FUNCTION_BLOCK "KistlerPresser _FB"   // FB2300, SCL
{ S7_Optimized_Access := 'FALSE' }
// stored: AutoNumber false, SetENOAutomatically false
   VAR_INPUT
      iHW_ID_Input : HW_SUBMODULE;
      iHW_ID_Output : HW_SUBMODULE;
      iSafetyInterlock : Bool;
      iContinueInterlock : Bool;
      iFltQuit : Bool;
      iSnEnable : Bool;   // True->Send SN
      iJogSpeed : Real;
      iJogMaxForce : Real;
      iCalibForce : Real;
      iXEncReference : Real;
      iReadIdentifier : Any;
      iReadPressData : Any;
      iWriteIdentifier : Any;
      iWritePressData : Any;
      iSpareByte : Array[0..19] of Byte;
   END_VAR
   VAR_OUTPUT
      oFltNo : Word;
      oError : Bool;
      oReady : Bool;
      oRdyAmp : Bool;
      oRdyCmd : Bool;
      oZeroXOk : Bool;
      oSetXRefOk : Bool;
      oHomeOk : Bool;
      oStartCycleOk : Bool;
      oCycleOK : Bool;
      oCycleNOK : Bool;
      oWaitRequest : Bool;
      oInHomePos : Bool;
      oRunSeq : Bool;
      oActProgNo : Int;
      oActLabelID : Int;
      oActSensorPos : Real;
      oActServoPos : Real;
      oActForce : Real;
      oActXEncRefValue : Real;
   END_VAR
   VAR
      ProgNo : Int;
      SelectSeq : Int;
      ZeroX : Bool;
      SetXRef : Bool;
      Homing : Bool;
      StartCycle : Bool;
      ContinueSeq : Bool;
      JogPos : Bool;
      JogNeg : Bool;
      JogPosActive : Bool;
      JogNegActive : Bool;
      SpareByte : Array[0..67] of Byte;
      InputMessages : Struct   // Status Inputs
         StatusBits : Struct
            "MIRROR-START" : Bool;   // Mirrored cycle START
            "MIRROR-TARE-Y" : Bool;   // Mirrored channel Y Tare or Reset Piezo
            "MIRROR-ZERO X" : Bool;   // Mirrored channel X Zeros
            "MIRROR-STEST-X" : Bool;   // Mirrored sensor test for sensor X
            "MIRROR-STEST-Y" : Bool;   // Mirrored sensor test for sensor Y
            "ReservedBit000.5" : Bool;   // Reserved
            "MASTER-MEAS" : Bool;   // Mirrored master measurement
            "INC-ZERO" : Bool;   // Mirrored zeros incremental sensor
            "ReservedBit001.0" : Bool;   // Reserved
            "MIRROR-ACK-ADMIN" : Bool;   // Mirrored acknowledgment with administrative rights (e.g.,corresponding warning, alarm)
            "ReservedBit001.2" : Bool;   // Reserved
            "MIRROR-ACCESS" : Bool;   // MIRROR-ACCESS
            AUTO : Bool;   // Mirrored production mode, no editing of setup is possible
            "STAT-RESET" : Bool;   // Mirrored statistics reset
            "STAT-DISABLE" : Bool;   // Deactivate mirrored statistics
            "TARE-EXTENDED-Y" : Bool;   // Mirrored Ext. channel Y Tare or Reset Piezo (maXYmos NC)
            MP : Byte;   // Mirrored measurement program choice
            "ReservedBit003.0" : Bool;   // Reserved
            "ReservedBit003.1" : Bool;   // Reserved
            "RESET-SN-GENERATOR" : Bool;   // Mirrored resetting of global serial number
            "ReservedBit003.3" : Bool;   // Reserved
            "ReservedBit003.4" : Bool;   // Reserved
            "BREAKETEST-ACTIVE" : Bool;   // Brake test is performed
            "ReservedBit003.6" : Bool;   // Reserved
            "ReservedBit003.7" : Bool;   // Reserved
            UNI : Byte;   // Mirrored input signals of UNI
            ReservedByte005 : Byte;   // Reserved
            READY : Bool;   // Already
            "OK-TOTAL" : Bool;   // Results GOOD
            "NOK-TOTAL" : Bool;   // Results BAD
            "NO-PASS" : Bool;   // NO-PASS exceeded
            "ReservedBit006.4" : Bool;   // Reserved
            "ReservedBit006.5" : Bool;   // Reserved
            WARN : Bool;   // Warning
            ALARM : Bool;   // Alarm
            S1 : Bool;   // Switching signal S1
            S2 : Bool;   // Switching signal S2
            "ReservedBit007.2" : Bool;   // Reserved
            "ReservedBit007.3" : Bool;   // Reserved
            "ReservedBit007.4" : Bool;   // Reserved
            "ReservedBit007.5" : Bool;   // Reserved
            "ReservedBit007.6" : Bool;   // Reserved
            "ReservedBit007.7" : Bool;   // Reserved
            "O-UNI" : Byte;   // Freely configurable output signal
            "DRIVE-ENABLE" : Bool;   // Mirrored enable drive
            "RUN-SEQUENCE" : Bool;   // Mirrored command process of the sequence
            "DRIVE-TO-HOMEPOS" : Bool;   // Mirrored command movement on base setting (MP-specific)
            "DRIVE-TO-REFPOS" : Bool;   // Mirrored command movement to reference position (global)
            "JOG-FW" : Bool;   // Mirrored command jogging forwards
            "JOG-BW" : Bool;   // Mirrored command jogging backwards
            "WAIT-REQUEST" : Bool;   // Output is set through sequence object Wait. Sequence waits for continuation through acknowledgment.
            "BRAKETEST-DONE" : Bool;   // Brake test performed.
            "SEQUENCE-STOPPED" : Bool;   // Sequence/command stopped
            "SEQUENCE-END" : Bool;   // Sequence/command ended
            "ONLINE-EO-NOK" : Bool;   // NOK for online evaluation of a corresponding EOs. Measurement ends.
            "EXT-STOP" : Bool;   // External stop was set in sequence object
            "SEQUENCE-ERROR" : Bool;   // Sequence/command error
            "DRIVE-ENABLED" : Bool;   // Enable drive set (current status of the enable)
            "HOMEPOS-REACHED" : Bool;   // Home position reached (NC joining module is in MP-specific home position)
            "REFPOS-REACHED" : Bool;   // Reference position reached (NC joining module is in global reference position)
            STANDSTILL : Bool;   // Standstill
            "BRAKETEST-REQ" : Bool;   // Brake test required
            "SERVO-WARN" : Bool;   // Warning message on the servo amplifier pending
            "SERVO-ERROR" : Bool;   // Alarm message on the servo amplifier pending
            "SMES-ACTIVE" : Bool;   // Safety status SMES active
            "SMST2-ACTIVE" : Bool;   // Safety status SMST2 active
            "SMM1-ACTIVE" : Bool;   // Safety status SMM1 active
            "USER-MODE-ACTIVE" : Bool;   // Output is active (1) when the monitoring of the control via the monitor (in the menu 'Service/Jog Mode' ... Sequence Mode... Referencing) is directly performed by the operator.
            SEQUENCE : Byte;   // Mirrored selection sequence Main, Sub1 ... 3
            "LABEL-ID" : Byte;   // Index of the cuurent trademark
            "CFG-MP" : Byte;   // Selecting of the measuring program for the transmission of data is intended. This applies to both writing and reading. See note below. If objects are to be interpreted globally, Byte 15.7 must be set.
            "ReservedBit015.0" : Bool;   // Reserved
            "ReservedBit015.1" : Bool;   // Reserved
            "ReservedBit015.2" : Bool;   // Reserved
            "ReservedBit015.3" : Bool;   // Reserved
            "ReservedBit015.4" : Bool;   // Reserved
            "ReservedBit015.5" : Bool;   // Reserved
            "ReservedBit015.6" : Bool;   // Reserved
            "GLOBAL-CFG-MP" : Bool;   // If this bit is set, the telegram data is interpreted as global objects.
            "MIRRIR-CFG-ADR" : Byte;   // Mirror CFG-ADR (up V 1.2.x.)
            "MIRRIR-CFG-LENGTH" : Byte;   // Mirror CFG-LENGTH (up V 1.2.x.)
            "SELECT-PAGE" : Byte;   // Selection of the page that is displayed in the address range from address 20.
            "TRANSMISSION-FAULT" : Bool;   // Error flag for transmission error. This is set upon detection of a transmission error with clearing of the bit ACK.
            ACK : Bool;   // Confirmation flag is set (= 1 byte 19.1) when maXYmos the desired action, which was triggered by the bit strobe executes.After receiving Bit ACK, Bit Strobe can be cleared. With clearing of bit strobe, bit ACK bit is reset.
            "DEVICE-AVAILABLE" : Bool;   // Wenn Bit gesetzt ist, ist das maXYmos Gerät über den Feldbus ansprechbar. Das Bit wird nach dem Gerätestart gesetzt und bleibt im Betrieb dauerhaft erhalten
            "ReservedBit019.3" : Bool;   // Reserved
            "CHANGEDSELECTED-MP" : Bool;   // Change flags of the measurement program changed. Flag isset (= 1) when it is detected that data has been modified in the measurement program since the last measurement. The flag is set after the measurement.
            "ReservedBit019.5" : Bool;   // Reserved
            "CHANGED--GLOBAL" : Bool;   // Change flags of global settings changed. Flag is set (= 1) when it has been recognized that global settings have been changed since the last measurement. Bit is only set if input bit is 19.6 = 0.
            "BACKUP-REQUEST" : Bool;   // Requirement to create a backup on the export server
         END_STRUCT;
         FreelyArea : Struct
            XEncRefValue : Real;
            CurValueX_1 : Real;
            CurValueX_2 : Real;
            CurValueY : Real;
            SerialNnmber { ExternalAccessible := 'False'; ExternalVisible := 'False'; ExternalWritable := 'False'} : Array[36..85] of Byte;
            "pvCurveXMIN-X" : Real;
            "pvCurveXMAX-X" : Real;
            "pvCurveYMIN-Y" : Real;
            "pvCurveYMAX-Y" : Real;
            PressData : Array[86..203] of Byte;
         END_STRUCT;
      END_STRUCT;
      OutputMessages : Struct   // Control Outputs
         ControlBits : Struct
            START : Bool;   // Cycle START
            "TARE-Y" : Bool;   // Channel Y Tare or Reset Piezo
            "ZERO X" : Bool;   // Channel X zeros
            "STEST-X" : Bool;   // Trigger sensor test for sensor X
            "STEST-Y" : Bool;   // Trigger sensor test for sensor Y
            "ReservedBit000.5" : Bool;   // Reserved
            "MASTER-MEAS" : Bool;   // MEAS Master measurement
            "INC-ZERO" : Bool;   // Zeros incremental sensor
            "ReservedBit001.0" : Bool;   // Reserved
            "ACK-ADMIN" : Bool;   // Acknowledgment with Admin rights (e.g., corresponding warning, alarm)
            "ReservedBit001.2" : Bool;   // Reserved
            ACCESS : Bool;   // Allows the PLC to give the operator access rights. The rights group (Setter, Operator, Admin) in effect is set via the protectionPlcLogon object. If ACCESS = 1, the operator can use these rights (does not have to register separately), when ACCESS = 0, this corresponds to a logoff.
            AUTO : Bool;   // Bit AUTO must be set (Byte 1.4 = 1) when the measurement program should be switched on using the PLC fieldbus. With AUTO = 1, the PLC has full control over maXYmo. A manual setup is thus also blocked!
            "STAT-RESET" : Bool;   // Rest statistics
            "STAT-DISABLE" : Bool;   // Deactivate statistics
            "TARE-EXTENDED-Y" : Bool;   // Ext. channel Y Tare or Reset Piezo (maXYmos NC)
            MP : Byte;   // Measurement program selection (see also byte 14 page control input control/config bits).
            "ReservedBit003.0" : Bool;   // Reserved
            "ReservedBit003.1" : Bool;   // Reserved
            "RESET-SN-GENERATOR" : Bool;   // Resetting of counter of global serial number
            "ReservedBit003.3" : Bool;   // Reserved
            "ReservedBit003.4" : Bool;   // Reserved
            "ReservedBit003.5" : Bool;   // Reserved
            "ReservedBit003.6" : Bool;   // Reserved
            "ReservedBit003.7" : Bool;   // Reserved
            UNI : Byte;   // Reserved for freely configurable digital input signals
            ReservedByte005 : Byte;   // Reserved
            ReservedByte006 : Byte;   // Reserved
            ReservedByte007 : Byte;   // Reserved
            ReservedByte008 : Byte;   // Reserved
            "DRIVE-ENABLE" : Bool;   // Release drive
            "RUN-SEQUENCE" : Bool;   // Command sequence has been run
            "DRIVE-TO-HOMEPOS" : Bool;   // Command movement to home position (MP-specific)
            "DRIVE-TO-REFPOS" : Bool;   // Command movement to reference position (global)
            "JOG-FW" : Bool;   // Command jogging forwards
            "JOG-BW" : Bool;   // Command jogging backwards
            "CONTNUEFROM-WAIT" : Bool;   // Continue command sequence after WAIT-REQUEST
            "MANUAL-BRAKETEST" : Bool;   // Perform command manual brake test
            "ReservedBit010.0" : Bool;   // Reserved
            "ReservedBit010.1" : Bool;   // Reserved
            "ReservedBit010.2" : Bool;   // Reserved
            "SEQ-EXT-STOP-REQ" : Bool;   // Externer Stop der Sequenz
            "ReservedBit010.4" : Bool;   // Reserved
            "ReservedBit010.5" : Bool;   // Reserved
            "ReservedBit010.6" : Bool;   // Reserved
            "ReservedBit010.7" : Bool;   // Reserved
            ReservedByte011 : Byte;   // Reserved
            "CURRENT SEQUENCE" : Byte;   // Select sequence main, Sub1 ... 3
            ReservedByte013 : Byte;   // Reserved
            "CFG-MP" : Byte;   // CFP Program number
            "ReservedBit015.0" : Bool;   // Reserved
            "ReservedBit015.1" : Bool;   // Reserved
            "ReservedBit015.2" : Bool;   // Reserved
            "ReservedBit015.3" : Bool;   // Reserved
            "ReservedBit015.4" : Bool;   // Reserved
            "ReservedBit015.5" : Bool;   // Reserved
            "ReservedBit015.6" : Bool;   // Reserved
            "GLOBAL-CFG-MP" : Bool;
            "CFG-ADDRESS" : Byte;
            "CFG-LENGTH" : Byte;
            "SELECT-PAGE" : Byte;
            "SAVE-TO-MP" : Bool;
            STROBE : Bool;
            "ReservedBit019.2" : Bool;   // Reserved
            "ReservedBit019.3" : Bool;   // Reserved
            "RESET-CHANGED-SELECTED-MP" : Bool;
            "ReservedBit019.5" : Bool;   // Reserved
            "RESET-CHANGEDGLOBAL" : Bool;
            "BACKUP-REQUEST" : Bool;
         END_STRUCT;
         FreelyArea : Struct
            XEncRefValue : Real;
            JogSpeed : Real;
            JogMaxForce : Real;
            CalibForce : Real;
            SerialNnmber { ExternalAccessible := 'False'; ExternalVisible := 'False'; ExternalWritable := 'False'} : Array[36..85] of Byte;
            PressData : Array[86..219] of Byte;
         END_STRUCT;
      END_STRUCT;
      Info : Struct
         ProgNo : Byte;
         SelectSeq : Byte;
         SelectPage : Byte;
         CfgAddress : Byte;
         CfgLength : Byte;
         Cancel : Bool;
         ContinueSeq : Bool;
      END_STRUCT;
      SetXRefRise : Bool;
      JogRise : Bool;
      HomingRise : Bool;
      StartCycleRise : Bool;
      FltQuitRise : Bool;
      SetXRefOld : Bool;
      JogOld : Bool;
      HomingOld : Bool;
      StartCycleOld : Bool;
      FltQuitOld : Bool;
      SetXRefAct : Bool;
      JogAct : Bool;
      HomeAct : Bool;
      CycleAct : Bool;
      OrderCount : Int;
      Index : Int;
      "Step" : Array[1..5] of Int;
      Ref_Timer_IN : Bool;
      JogTimer_IN : Bool;
      HomeTimer_IN : Bool;
      SeqTimer_IN : Bool;
      HomeTime : Time;
      SeqTime : Time;
      Ref_Timer { S7_SetPoint := 'True'} : TON_TIME;
      Jog_Timer { S7_SetPoint := 'True'} : TON_TIME;
      Home_Timer { S7_SetPoint := 'True'} : TON_TIME;
      Seq_Timer { S7_SetPoint := 'True'} : TON_TIME;
   END_VAR
   VAR_TEMP
      tmpSource : Byte;
      tmpRetVal : Int;
      pTempPNIOData : Any;
      pTempPressdata : Any;
      pAnyPressdata AT pTempPressdata : Struct
         SyntaxID : Byte;
         DataType : Byte;
         DataCount : Int;
         DBNumber : Word;
         BytePointer : DWord;
      END_STRUCT;
   END_VAR
BEGIN
   (*
   Kistler Presser Control Function Block
   ruhlamat Automation Technologies(Suzhou ) Co.,Ltd
   Copyright(c ) 2016.All rights reserved.
   -------------------------------------------------------------------------------------------
   NAME OF FUNCTION BLOCK:"maXYmosCtrl"
   FAMILY:ruhlamat PSL
   VERSION:V1.1
   AUTHOR:Chaoyao.Zheng
   LAST CHANGE:11.09.2017
   -------------------------------------------------------------------------------------------
   Date Name Activity
   11.09.2017 Chaoyao.Zheng Created(V1.0)
   12.21.2017 Qianfeng.Yang Update(Step7->TIA Portal)
   -------------------------------------------------------------------------------------------
   // F001: MEM not ready
   // F002: IndraDrive not ready
   // F003: User mode is active
   // F004: Order when FB not ready
   // F005: Several orders set at the same time
   // F006: Invalid program number
   // F007: Timeout when homing procedures 
   // F008: Timeout when press-in cycle
   // F009: Timeout data handshake
   // F010: Timeout when set var
   *)
   //Begin
   #pTempPNIOData := #InputMessages;
   #tmpRetVal := DPRD_DAT(LADDR := #iHW_ID_Input,
                          RECORD => #pTempPNIOData);
   IF #tmpRetVal <> 0 THEN
       GOTO Error;
   END_IF;

   #pTempPressdata := #iReadIdentifier;
   IF #pAnyPressdata.DataType = B#16#2 AND #pAnyPressdata.DataCount > 0 THEN
       #tmpRetVal := BLKMOV(SRCBLK := #InputMessages.FreelyArea.SerialNnmber, DSTBLK => #pTempPressdata);
   END_IF;

   #pTempPressdata := #iReadPressData;
   IF #pAnyPressdata.DataType = B#16#2 AND #pAnyPressdata.DataCount > 0 THEN
       #tmpRetVal := BLKMOV(SRCBLK := #InputMessages.FreelyArea.PressData, DSTBLK => #pTempPressdata);
   END_IF;

   #oActXEncRefValue := #InputMessages.FreelyArea.XEncRefValue;
   #oActProgNo := BYTE_TO_INT(#InputMessages.StatusBits.MP);
   #oActLabelID := BYTE_TO_INT(#InputMessages.StatusBits."LABEL-ID");
   #oActSensorPos := #InputMessages.FreelyArea.CurValueX_1;
   #oActServoPos := #InputMessages.FreelyArea.CurValueX_2;
   #oActForce := #InputMessages.FreelyArea.CurValueY;
   #oInHomePos := #InputMessages.StatusBits."HOMEPOS-REACHED";
   #oRunSeq := #InputMessages.StatusBits."RUN-SEQUENCE";
   #JogPosActive := #InputMessages.StatusBits."JOG-FW";
   #JogNegActive := #InputMessages.StatusBits."JOG-BW";

   IF #iSafetyInterlock AND NOT #InputMessages.StatusBits."SMES-ACTIVE" THEN
       #oRdyAmp := #InputMessages.StatusBits."DRIVE-ENABLED";
       #OutputMessages.ControlBits."DRIVE-ENABLE" := TRUE;
   ELSE
       #oRdyAmp := FALSE;
       #OutputMessages.ControlBits."DRIVE-ENABLE" := FALSE;
   END_IF;

   #FltQuitRise := NOT #FltQuitOld AND #iFltQuit;
   #FltQuitOld := #iFltQuit;
   #SetXRefRise := NOT #SetXRefOld AND #SetXRef;
   #SetXRefOld := #SetXRef;
   #HomingRise := NOT #HomingOld AND #Homing;
   #HomingOld := #Homing;
   #JogRise := NOT #JogOld AND (#JogPos OR #JogNeg);
   #JogOld := #JogPos OR #JogNeg;
   #StartCycleRise := NOT #StartCycleOld AND #StartCycle;
   #StartCycleOld := #StartCycle;

   IF #FltQuitRise THEN
       IF #OrderCount = 0 THEN
           #oFltNo := W#16#0000;
       END_IF;
       #OutputMessages.ControlBits."ACK-ADMIN" := TRUE;
   ELSE
       #OutputMessages.ControlBits."ACK-ADMIN" := FALSE;
   END_IF;

   IF NOT #InputMessages.StatusBits."DEVICE-AVAILABLE" OR #InputMessages.StatusBits.ALARM THEN
       IF #oFltNo = W#16#0000 THEN
           #oFltNo := W#16#F001;
       END_IF;
   END_IF;

   IF #InputMessages.StatusBits."SERVO-ERROR" THEN
       IF #oFltNo = W#16#0000 THEN
           #oFltNo := W#16#F002;
       END_IF;
   END_IF;

   IF #InputMessages.StatusBits."USER-MODE-ACTIVE" THEN
       IF #oFltNo = W#16#0000 THEN
           #oFltNo := W#16#F003;
       END_IF;
   END_IF;

   IF #oFltNo = W#16#0000 THEN
       IF #JogRise OR #HomingRise OR #StartCycleRise THEN
           IF NOT #oRdyCmd THEN
               #oFltNo := W#16#F004;
           END_IF;
       END_IF;
   END_IF;

   #OrderCount := 0;
   IF #JogPos OR #JogNeg THEN
       #OrderCount := #OrderCount + 1;
   END_IF;

   IF #Homing THEN
       #OrderCount := #OrderCount + 1;
   END_IF;

   IF #StartCycle THEN
       #OrderCount := #OrderCount + 1;
   END_IF;

   IF #SetXRef THEN
       #OrderCount := #OrderCount + 1;
   END_IF;

   IF #OrderCount > 1 THEN
       IF #oFltNo = W#16#0000 THEN
           #oFltNo := W#16#F005;
       END_IF;
   END_IF;

   IF (#oFltNo = W#16#0000)
   THEN
       IF (#ProgNo < 0) OR
           (#ProgNo > 127)
       THEN
           #oFltNo := W#16#F006;
       END_IF;
   END_IF;

   IF #oFltNo = W#16#0000 THEN
       IF #SelectSeq < 0 OR #SelectSeq > 3 THEN
           #oFltNo := W#16#F006;
       END_IF;
   END_IF;

   // ***********************************************************************
   // Sequence --- SetXRef
   // ***********************************************************************
   #Index := 1;
   IF NOT #SetXRef THEN
       IF #SetXRefAct THEN
           #OutputMessages.ControlBits.STROBE := FALSE;
           #SetXRefAct := FALSE;
       END_IF;
   END_IF;

   IF #oFltNo = W#16#0000 AND #SetXRefRise THEN
       #Info.ProgNo := INT_TO_BYTE(#ProgNo);
       #Info.SelectSeq := INT_TO_BYTE(#SelectSeq);
       #Info.SelectPage := 0;
       #Info.CfgAddress := 0;
       #Info.CfgLength := 4;
       #SetXRefAct := TRUE;
       #oSetXRefOk := FALSE;
       #Step[#Index] := 0;
   END_IF;

   #Ref_Timer_IN := FALSE;
   IF #SetXRefAct THEN
       CASE #Step[#Index] OF
           0:
               #Ref_Timer_IN := FALSE;
               #Step[#Index] := #Step[#Index] + 1;

           1:
               IF #InputMessages.StatusBits.READY THEN
                   #Ref_Timer_IN := FALSE;
                   #OutputMessages.ControlBits."CFG-MP" := #Info.ProgNo;
                   #OutputMessages.ControlBits."SELECT-PAGE" := #Info.SelectPage;
                   #OutputMessages.ControlBits."CFG-ADDRESS" := #Info.CfgAddress;
                   #OutputMessages.ControlBits."CFG-LENGTH" := #Info.CfgLength;
                   #OutputMessages.ControlBits."SAVE-TO-MP" := TRUE;
                   #Step[#Index] := #Step[#Index] + 1;
               ELSE
                   #Ref_Timer_IN := TRUE;
                   IF #Ref_Timer.Q THEN
                       #Ref_Timer_IN := FALSE;
                       #oFltNo := W#16#F011;
                       #Step[#Index] := 99;

                   END_IF;
               END_IF;

           2:
               IF #InputMessages.StatusBits."CFG-MP" = #Info.ProgNo AND #InputMessages.StatusBits."SELECT-PAGE" = #Info.SelectPage AND #InputMessages.StatusBits."MIRRIR-CFG-ADR" = #Info.CfgAddress AND #InputMessages.StatusBits."MIRRIR-CFG-LENGTH" = #Info.CfgLength THEN
                   #Ref_Timer_IN := FALSE;
                   #OutputMessages.ControlBits.STROBE := TRUE;
                   #Step[#Index] := #Step[#Index] + 1;
               ELSE
                   #Ref_Timer_IN := TRUE;
                   IF #Ref_Timer.Q THEN
                       #Ref_Timer_IN := FALSE;
                       #oFltNo := W#16#F012;
                       #Step[#Index] := 99;
                   END_IF;
               END_IF;

           3:
               IF #InputMessages.StatusBits.ACK THEN
                   #Ref_Timer_IN := FALSE;
                   IF #InputMessages.StatusBits."TRANSMISSION-FAULT" THEN
                       #oFltNo := W#16#F013;
                   ELSE
                       #OutputMessages.ControlBits.STROBE := FALSE;
                       #Step[#Index] := 99;
                   END_IF;
               ELSE
                   #Ref_Timer_IN := TRUE;
                   IF #Ref_Timer.Q THEN
                       #Ref_Timer_IN := FALSE;
                       #oFltNo := W#16#F014;
                       #Step[#Index] := 99;
                   END_IF;
               END_IF;

           99:
               #Ref_Timer_IN := FALSE;
               #OutputMessages.ControlBits.STROBE := FALSE;
               #SetXRefAct := FALSE;
               IF #oFltNo = W#16#0000 THEN
                   #oSetXRefOk := TRUE;
               END_IF;

           ELSE
               ;
       END_CASE;
   END_IF;
   #Ref_Timer(IN := #Ref_Timer_IN,
              PT := t#1s);

   // ***********************************************************************
   // Sequence --- Jog Pos/Neg
   // ***********************************************************************
   #Index := 2;
   IF NOT #JogPos AND NOT #JogNeg THEN
       IF #JogAct THEN
           #Info.Cancel := TRUE;
       END_IF;
   END_IF;

   IF #oFltNo = W#16#0000 AND #JogRise THEN
       #Info.ProgNo := INT_TO_BYTE(#ProgNo);
       #Info.SelectSeq := INT_TO_BYTE(#SelectSeq);
       #Info.SelectPage := 0;
       #Info.CfgAddress := 4;
       #Info.CfgLength := 8;
       #JogAct := TRUE;
       #Step[#Index] := 0;
   END_IF;

   #JogTimer_IN := FALSE;
   IF #JogAct THEN
       CASE #Step[#Index] OF
           0:
               #JogTimer_IN := FALSE;
               #Step[#Index] := #Step[#Index] + 1;

           1:
               IF #InputMessages.StatusBits.READY THEN
                   #JogTimer_IN := FALSE;
                   #OutputMessages.ControlBits."CFG-MP" := #Info.ProgNo;
                   #OutputMessages.ControlBits."SELECT-PAGE" := #Info.SelectPage;
                   #OutputMessages.ControlBits."CFG-ADDRESS" := #Info.CfgAddress;
                   #OutputMessages.ControlBits."CFG-LENGTH" := #Info.CfgLength;
                   #OutputMessages.ControlBits."SAVE-TO-MP" := FALSE;
                   #Step[#Index] := #Step[#Index] + 1;
               ELSE
                   #JogTimer_IN := TRUE;
                   IF #Jog_Timer.Q THEN
                       #JogTimer_IN := FALSE;
                       #oFltNo := W#16#F008;
                       #Step[#Index] := 99;
                   END_IF;
               END_IF;

           2:
               IF #InputMessages.StatusBits."CFG-MP" = #Info.ProgNo AND #InputMessages.StatusBits."SELECT-PAGE" = #Info.SelectPage AND #InputMessages.StatusBits."MIRRIR-CFG-ADR" = #Info.CfgAddress AND #InputMessages.StatusBits."MIRRIR-CFG-LENGTH" = #Info.CfgLength THEN
                   #JogTimer_IN := FALSE;
                   #OutputMessages.ControlBits.STROBE := TRUE;
                   #Step[#Index] := #Step[#Index] + 1;
               ELSE
                   #JogTimer_IN := TRUE;
                   IF #Jog_Timer.Q THEN
                       #JogTimer_IN := FALSE;
                       #oFltNo := W#16#F008;
                       #Step[#Index] := 99;
                   END_IF;
               END_IF;

           3:
               IF #InputMessages.StatusBits.ACK THEN
                   #JogTimer_IN := FALSE;
                   IF #InputMessages.StatusBits."TRANSMISSION-FAULT" THEN
                       #oFltNo := W#16#F008;
                   ELSE
                       #OutputMessages.ControlBits.STROBE := FALSE;
                       #Step[#Index] := #Step[#Index] + 1;
                   END_IF;
               ELSE
                   #JogTimer_IN := TRUE;
                   IF #Jog_Timer.Q THEN
                       #JogTimer_IN := FALSE;
                       #oFltNo := W#16#F008;
                       #Step[#Index] := 99;
                   END_IF;
               END_IF;

           4:
               #Step[#Index] := #Step[#Index] + 1;

           5:
               IF #InputMessages.StatusBits."DRIVE-ENABLED" THEN
                   #JogTimer_IN := FALSE;
                   #Step[#Index] := #Step[#Index] + 1;
               ELSE
                   #JogTimer_IN := TRUE;
                   IF #Jog_Timer.Q THEN
                       #JogTimer_IN := FALSE;
                       #oFltNo := W#16#F007;
                       #Step[#Index] := 99;
                   END_IF;
               END_IF;

           6:
               IF #JogPos AND NOT #JogNeg THEN
                   #OutputMessages.ControlBits."JOG-FW" := TRUE;
                   #OutputMessages.ControlBits."JOG-BW" := FALSE;
               ELSIF NOT #JogPos AND #JogNeg THEN
                   #OutputMessages.ControlBits."JOG-FW" := FALSE;
                   #OutputMessages.ControlBits."JOG-BW" := TRUE;
               ELSE
                   #Step[#Index] := 99;
               END_IF;

           99:
               #JogTimer_IN := FALSE;
               #OutputMessages.ControlBits.STROBE := FALSE;
               #OutputMessages.ControlBits."JOG-FW" := FALSE;
               #OutputMessages.ControlBits."JOG-BW" := FALSE;
               #JogAct := FALSE;

           ELSE
               ;

       END_CASE;
   END_IF;
   #Jog_Timer(IN := #JogTimer_IN,
              PT := T#1s);

   // ***********************************************************************
   // Sequence --- Drive to home position
   // ***********************************************************************
   #Index := 3;

   IF NOT #Homing THEN
       #oHomeOk := FALSE;
       IF #HomeAct THEN
           #OutputMessages.ControlBits.STROBE := FALSE;
           #OutputMessages.ControlBits.AUTO := FALSE;
           #OutputMessages.ControlBits."DRIVE-TO-HOMEPOS" := FALSE;
           #OutputMessages.ControlBits."DRIVE-TO-REFPOS" := FALSE;
           #HomeAct := FALSE;
       END_IF;
   END_IF;

   //IF #oFltNo = W#16#0000 AND #HomingRise THEN
   //#InputMessages.StatusBits.READY AND 
   IF #InputMessages.StatusBits.READY AND #HomingRise AND NOT #InputMessages.StatusBits.ALARM AND NOT #InputMessages.StatusBits.WARN THEN
       #Info.ProgNo := INT_TO_BYTE(#ProgNo);
       #HomeAct := TRUE;
       #oHomeOk := FALSE;
       #Step[#Index] := 0;
   END_IF;

   #HomeTimer_IN := FALSE;
   IF #HomeAct THEN
       CASE #Step[#Index] OF
           0:
               #HomeTimer_IN := FALSE;
               #HomeTime := t#1S;
               #Step[#Index] := #Step[#Index] + 1;

           1:
               //  IF #InputMessages.StatusBits.READY THEN
               IF #InputMessages.StatusBits.READY AND NOT #InputMessages.StatusBits.ALARM AND NOT #InputMessages.StatusBits.WARN THEN
                   #HomeTimer_IN := FALSE;
                   #OutputMessages.ControlBits.AUTO := TRUE;
                   #Step[#Index] := #Step[#Index] + 1;
               ELSE
                   #HomeTimer_IN := TRUE;
                   #HomeTime := t#1S;
                   IF #Home_Timer.Q THEN
                       #HomeTimer_IN := FALSE;
                       #oFltNo := W#16#F008;
                       #Step[#Index] := 99;
                   END_IF;
               END_IF;

           2:
               IF #InputMessages.StatusBits.READY AND #InputMessages.StatusBits.AUTO THEN
                   #HomeTimer_IN := FALSE;
                   #OutputMessages.ControlBits.MP := #Info.ProgNo;
                   #Step[#Index] := #Step[#Index] + 1;
               ELSE
                   #HomeTimer_IN := TRUE;
                   #HomeTime := t#1S;
                   IF #Home_Timer.Q THEN
                       #HomeTimer_IN := FALSE;
                       #oFltNo := W#16#F008;
                       #Step[#Index] := 99;
                   END_IF;
               END_IF;

           3:
               IF #InputMessages.StatusBits.MP = #Info.ProgNo THEN
                   #HomeTimer_IN := FALSE;
                   #OutputMessages.ControlBits.AUTO := FALSE;
                   #Step[#Index] := #Step[#Index] + 1;
               ELSE
                   #HomeTimer_IN := TRUE;
                   #HomeTime := t#1S;
                   IF #Home_Timer.Q THEN
                       #HomeTimer_IN := FALSE;
                       #oFltNo := W#16#F008;
                       #Step[#Index] := 99;
                   END_IF;
               END_IF;

           4:
               IF NOT #InputMessages.StatusBits.AUTO THEN
                   #HomeTimer_IN := FALSE;
                   #Step[#Index] := #Step[#Index] + 1;
               ELSE
                   #HomeTimer_IN := TRUE;
                   #HomeTime := t#1S;
                   IF #Home_Timer.Q THEN
                       #HomeTimer_IN := FALSE;
                       #oFltNo := W#16#F008;
                       #Step[#Index] := 99;
                   END_IF;
               END_IF;

           5:
               IF #InputMessages.StatusBits."HOMEPOS-REACHED" THEN
                   #Step[#Index] := 99;
               ELSIF #InputMessages.StatusBits."DRIVE-ENABLED" AND NOT #InputMessages.StatusBits."SEQUENCE-STOPPED" AND NOT #InputMessages.StatusBits."HOMEPOS-REACHED" THEN
                   #HomeTimer_IN := FALSE;
                   #OutputMessages.ControlBits."DRIVE-TO-HOMEPOS" := TRUE;
                   #Step[#Index] := #Step[#Index] + 1;
               ELSE
                   ;
                   #HomeTimer_IN := TRUE;
                   #HomeTime := t#2S;
                   IF #Home_Timer.Q THEN
                       #HomeTimer_IN := FALSE;
                       #oFltNo := W#16#F007;
                       #Step[#Index] := 99;
                   END_IF;
               END_IF;

           6:
               IF #InputMessages.StatusBits."DRIVE-TO-HOMEPOS" THEN
                   #HomeTimer_IN := FALSE;
                   #Step[#Index] := #Step[#Index] + 1;
               ELSE
                   ;
                   #HomeTimer_IN := TRUE;
                   #HomeTime := t#2S;
                   IF #Home_Timer.Q THEN
                       #HomeTimer_IN := FALSE;
                       #oFltNo := W#16#F007;
                       #Step[#Index] := 99;
                   END_IF;
               END_IF;

           7:
               IF #InputMessages.StatusBits."HOMEPOS-REACHED" THEN
                   #HomeTimer_IN := FALSE;
                   #OutputMessages.ControlBits."DRIVE-TO-HOMEPOS" := FALSE;
                   #Step[#Index] := #Step[#Index] + 1;
               ELSE
                   ;
                   #HomeTimer_IN := TRUE;
                   #HomeTime := t#60S;
                   IF #Home_Timer.Q THEN
                       #HomeTimer_IN := FALSE;
                       #oFltNo := W#16#F007;
                       #Step[#Index] := 99;
                   END_IF;
               END_IF;

           8:
               IF NOT #InputMessages.StatusBits."DRIVE-TO-HOMEPOS" THEN
                   #HomeTimer_IN := FALSE;
                   #Step[#Index] := 99;
               ELSE
                   #HomeTimer_IN := TRUE;
                   #HomeTime := t#2S;
                   IF #Home_Timer.Q THEN
                       #HomeTimer_IN := FALSE;
                       #oFltNo := W#16#F007;
                       #Step[#Index] := 99;
                   END_IF;
               END_IF;

           99:
               #HomeTimer_IN := FALSE;
               #OutputMessages.ControlBits.STROBE := FALSE;
               #OutputMessages.ControlBits.AUTO := FALSE;
               #OutputMessages.ControlBits."DRIVE-TO-HOMEPOS" := FALSE;
               #OutputMessages.ControlBits."DRIVE-TO-REFPOS" := FALSE;

               #HomeAct := FALSE;
               IF #oFltNo = W#16#0000 THEN
                   #oHomeOk := TRUE;
               END_IF;

           ELSE
               ;

       END_CASE;
   END_IF;
   #Home_Timer(IN := #HomeTimer_IN,
               PT := #HomeTime);


   // ***********************************************************************
   // Sequence --- Sequence mode
   // ***********************************************************************
   #Index := 4;
   IF NOT #StartCycle THEN
       #oStartCycleOk := FALSE;
       IF #CycleAct THEN
           #OutputMessages.ControlBits.AUTO := FALSE;
           #OutputMessages.ControlBits.STROBE := FALSE;
           #OutputMessages.ControlBits."RUN-SEQUENCE" := FALSE;
           #OutputMessages.ControlBits."CONTNUEFROM-WAIT" := FALSE;
           #CycleAct := FALSE;
       END_IF;
   END_IF;


   IF #oFltNo = W#16#0000 AND #StartCycleRise THEN
       #Info.ProgNo := INT_TO_BYTE(#ProgNo);
       #Info.SelectSeq := INT_TO_BYTE(#SelectSeq);
       #Info.SelectPage := 0;
       #Info.CfgAddress := 16;
       #pTempPressdata := #iWritePressData;
       #Info.CfgLength := INT_TO_BYTE(#pAnyPressdata.DataCount) + 50;
       #CycleAct := TRUE;
       #oStartCycleOk := FALSE;
       #oCycleOK := FALSE;
       #oCycleNOK := FALSE;
       #Step[#Index] := 0;
       #Step[#Index + 1] := 0;
       IF #Info.SelectSeq = 0 THEN
           #tmpRetVal := BLKMOV(SRCBLK := #iWriteIdentifier,
                                DSTBLK => #OutputMessages.FreelyArea.SerialNnmber);
           #tmpRetVal := BLKMOV(SRCBLK := #iWritePressData,
                                DSTBLK => #OutputMessages.FreelyArea.PressData);
       END_IF;
   END_IF;

   #oWaitRequest := #InputMessages.StatusBits."WAIT-REQUEST";
   #OutputMessages.ControlBits."CONTNUEFROM-WAIT" := #ContinueSeq AND #iContinueInterlock;

   #SeqTimer_IN := FALSE;
   IF #CycleAct THEN
       CASE #Step[#Index] OF
           0:
               #SeqTimer_IN := FALSE;
               IF #iSnEnable THEN
                   #Step[#Index] := #Step[#Index] + 1;
               ELSE
                   #Step[#Index] := 5;
               END_IF;

           1:
               IF #InputMessages.StatusBits.READY THEN
                   #SeqTimer_IN := FALSE;
                   #OutputMessages.ControlBits."CFG-MP" := #Info.ProgNo;
                   #OutputMessages.ControlBits."SELECT-PAGE" := #Info.SelectPage;
                   #OutputMessages.ControlBits."CFG-ADDRESS" := #Info.CfgAddress;
                   #OutputMessages.ControlBits."CFG-LENGTH" := #Info.CfgLength;
                   #OutputMessages.ControlBits."SAVE-TO-MP" := FALSE;
                   #Step[#Index] := #Step[#Index] + 1;
               ELSE
                   ;
                   #SeqTimer_IN := TRUE;
                   #SeqTime := T#1S;
                   IF #Seq_Timer.Q THEN
                       #SeqTimer_IN := FALSE;
                       #oFltNo := W#16#F008;
                       #Step[#Index] := 99;
                   END_IF;
               END_IF;

           2:
               IF #InputMessages.StatusBits."CFG-MP" = #Info.ProgNo AND #InputMessages.StatusBits."SELECT-PAGE" = #Info.SelectPage AND #InputMessages.StatusBits."MIRRIR-CFG-ADR" = #Info.CfgAddress AND #InputMessages.StatusBits."MIRRIR-CFG-LENGTH" = #Info.CfgLength THEN
                   #SeqTimer_IN := FALSE;
                   #OutputMessages.ControlBits.STROBE := TRUE;
                   #Step[#Index] := #Step[#Index] + 1;
               ELSE
                   ;
                   #SeqTimer_IN := TRUE;
                   #SeqTime := T#1S;
                   IF #Seq_Timer.Q THEN
                       #SeqTimer_IN := FALSE;
                       #oFltNo := W#16#F008;
                       #Step[#Index] := 99;
                   END_IF;
               END_IF;

           3:
               IF #InputMessages.StatusBits.ACK THEN
                   #SeqTimer_IN := FALSE;
                   IF #InputMessages.StatusBits."TRANSMISSION-FAULT" THEN
                       #oFltNo := W#16#F008;
                   ELSE
                       #OutputMessages.ControlBits.STROBE := FALSE;
                       #Step[#Index] := #Step[#Index] + 1;
                   END_IF;
               ELSE
                   ;
                   #SeqTimer_IN := TRUE;
                   #SeqTime := T#1S;
                   IF #Seq_Timer.Q THEN
                       #SeqTimer_IN := FALSE;
                       #oFltNo := W#16#F008;
                       #Step[#Index] := 99;
                   END_IF;
               END_IF;

           4:
               #Step[#Index] := #Step[#Index] + 1;

           5:
               IF #InputMessages.StatusBits.READY THEN
                   #SeqTimer_IN := FALSE;
                   #OutputMessages.ControlBits.AUTO := TRUE;
                   #Step[#Index] := #Step[#Index] + 1;
               ELSE
                   ;
                   #SeqTimer_IN := TRUE;
                   #SeqTime := T#1S;
                   IF #Seq_Timer.Q THEN
                       #SeqTimer_IN := FALSE;
                       #oFltNo := W#16#F008;
                       #Step[#Index] := 99;
                   END_IF;
               END_IF;

           6:
               IF #InputMessages.StatusBits."DRIVE-ENABLED" AND NOT #InputMessages.StatusBits."SEQUENCE-STOPPED" AND #InputMessages.StatusBits.READY AND #InputMessages.StatusBits.AUTO THEN
                   #SeqTimer_IN := FALSE;
                   #OutputMessages.ControlBits.MP := #Info.ProgNo;
                   #OutputMessages.ControlBits."CURRENT SEQUENCE" := #Info.SelectSeq;
                   #Step[#Index] := #Step[#Index] + 1;
               ELSE
                   ;
                   #SeqTimer_IN := TRUE;
                   #SeqTime := T#1S;
                   IF #Seq_Timer.Q THEN
                       #SeqTimer_IN := FALSE;
                       #oFltNo := W#16#F008;
                       #Step[#Index] := 99;
                   END_IF;
               END_IF;

           7:
               IF #InputMessages.StatusBits.MP = #Info.ProgNo AND #InputMessages.StatusBits.SEQUENCE = #Info.SelectSeq THEN
                   #SeqTimer_IN := FALSE;
                   #OutputMessages.ControlBits."RUN-SEQUENCE" := TRUE;
                   #Step[#Index] := #Step[#Index] + 1;
               ELSE
                   ;
                   #SeqTimer_IN := TRUE;
                   #SeqTime := T#1S;
                   IF #Seq_Timer.Q THEN
                       #SeqTimer_IN := FALSE;
                       #oFltNo := W#16#F008;
                       #Step[#Index] := 99;
                   END_IF;
               END_IF;

           8:
               IF #InputMessages.StatusBits."RUN-SEQUENCE" AND NOT #InputMessages.StatusBits."SEQUENCE-END" AND #InputMessages.StatusBits."DRIVE-ENABLED" AND NOT #InputMessages.StatusBits.WARN AND NOT #InputMessages.StatusBits.ALARM THEN
                   #SeqTimer_IN := FALSE;
                   #Step[#Index] := #Step[#Index] + 1;
               ELSE
                   ;
                   #SeqTimer_IN := TRUE;
                   #SeqTime := T#2S;
                   IF #Seq_Timer.Q THEN
                       #SeqTimer_IN := FALSE;
                       #oFltNo := W#16#F008;
                       #Step[#Index] := 99;
                   END_IF;
               END_IF;

           9:
               IF #InputMessages.StatusBits."SEQUENCE-STOPPED" AND #InputMessages.StatusBits."SEQUENCE-END" THEN
                   #SeqTimer_IN := FALSE;
                   #OutputMessages.ControlBits."RUN-SEQUENCE" := FALSE;
                   #Step[#Index] := #Step[#Index] + 1;
               ELSE
                   ;
                   #SeqTimer_IN := TRUE;
                   #SeqTime := T#20m;
                   IF #Seq_Timer.Q THEN
                       #SeqTimer_IN := FALSE;
                       #oFltNo := W#16#F008;
                       #Step[#Index] := 99;
                   END_IF;
               END_IF;

           10:
               IF NOT #InputMessages.StatusBits."RUN-SEQUENCE" AND NOT #InputMessages.StatusBits."SEQUENCE-STOPPED" THEN
                   #SeqTimer_IN := FALSE;
                   #Step[#Index] := 99;
               ELSE
                   ;
                   #SeqTimer_IN := TRUE;
                   #SeqTime := T#2S;
                   IF #Seq_Timer.Q THEN
                       #SeqTimer_IN := FALSE;
                       #oFltNo := W#16#F008;
                       #Step[#Index] := 99;
                   END_IF;
               END_IF;

           99:
               #SeqTimer_IN := FALSE;
               #OutputMessages.ControlBits.AUTO := FALSE;
               #OutputMessages.ControlBits.STROBE := FALSE;
               #OutputMessages.ControlBits."RUN-SEQUENCE" := FALSE;
               #OutputMessages.ControlBits."CONTNUEFROM-WAIT" := FALSE;
               #CycleAct := FALSE;
               IF #oFltNo = W#16#0000 THEN
                   #oStartCycleOk := TRUE;
               END_IF;
               #tmpSource := B#16#00;
               #tmpRetVal := FILL(BVAL := #tmpSource, BLK => #OutputMessages.FreelyArea.SerialNnmber);
               #tmpRetVal := FILL(BVAL := #tmpSource, BLK => #OutputMessages.FreelyArea.PressData);
           ELSE
               ;
       END_CASE;

       CASE #Step[#Index + 1] OF
           0:
               IF #InputMessages.StatusBits.READY AND #OutputMessages.ControlBits."RUN-SEQUENCE" THEN
                   #Step[#Index + 1] := 1;
               END_IF;

           1:
               IF NOT #InputMessages.StatusBits.READY THEN
                   #Step[#Index + 1] := 2;
               END_IF;

           2:
               IF #InputMessages.StatusBits.READY THEN
               (* Evaluation result *)
                   #oCycleOK := #InputMessages.StatusBits."OK-TOTAL" AND NOT #InputMessages.StatusBits."NOK-TOTAL";
                   #oCycleNOK := NOT #InputMessages.StatusBits."OK-TOTAL" OR #InputMessages.StatusBits."NOK-TOTAL";
                   #Step[#Index + 1] := 99;
               END_IF;

           ELSE
               ;

       END_CASE;
   END_IF;
   #Seq_Timer(IN := #SeqTimer_IN,
              PT := #SeqTime);

   IF #OrderCount <> 1 THEN
       #OutputMessages.ControlBits.AUTO := FALSE;
       #OutputMessages.ControlBits.STROBE := FALSE;
       #OutputMessages.ControlBits."RUN-SEQUENCE" := FALSE;
       #OutputMessages.ControlBits."CONTNUEFROM-WAIT" := FALSE;
       #OutputMessages.ControlBits."DRIVE-TO-HOMEPOS" := FALSE;
       #OutputMessages.ControlBits."DRIVE-TO-REFPOS" := FALSE;
       #OutputMessages.ControlBits."JOG-FW" := FALSE;
       #OutputMessages.ControlBits."JOG-BW" := FALSE;
   END_IF;
   IF #OrderCount = 0 THEN
       #OutputMessages.ControlBits.MP := INT_TO_BYTE(#ProgNo);
   END_IF;
   #oError := #oFltNo <> W#16#0000;
   #oReady := #oFltNo = W#16#000 AND #oRdyAmp;
   #oRdyCmd := #oFltNo = W#16#0000 AND #oRdyAmp AND NOT #JogAct AND NOT #HomeAct AND NOT #CycleAct AND NOT #SetXRefAct AND NOT #JogPos AND NOT #JogNeg AND NOT #Homing AND NOT #StartCycle AND NOT #SetXRef AND NOT #InputMessages.StatusBits."RUN-SEQUENCE";
   IF #oRdyCmd OR #InputMessages.StatusBits."WAIT-REQUEST" THEN
       #OutputMessages.ControlBits."ZERO X" := #ZeroX;
   ELSE
       #OutputMessages.ControlBits."ZERO X" := FALSE;
   END_IF;

   #oZeroXOk := #InputMessages.StatusBits."MIRROR-ZERO X";
   #OutputMessages.FreelyArea.XEncRefValue := #iXEncReference;
   #OutputMessages.FreelyArea.JogSpeed := #iJogSpeed;
   #OutputMessages.FreelyArea.JogMaxForce := #iJogMaxForce;
   #OutputMessages.FreelyArea.CalibForce := #iCalibForce;

   #pTempPNIOData := #OutputMessages;
   #tmpRetVal := DPWR_DAT(LADDR := #iHW_ID_Output,
                          RECORD := #pTempPNIOData);
   IF #tmpRetVal <> 0 THEN
       GOTO Error;
   END_IF;

   //End function block
   ENO := 1;
   RETURN;
   //Error
   Error:
   #oError := 1;
   ENO := 0;
   RETURN;
END_FUNCTION_BLOCK

FUNCTION "Robot" : Void   // FC2400, LAD
{ S7_Optimized_Access := 'TRUE' }
// stored: AutoNumber false, SetENOAutomatically false
   VAR_TEMP   // added for the SCL form of the ladder/FBD networks
      _w1 : Bool;
      _w2 : Bool;
      _w3 : Bool;
      _w4 : Bool;
      _w5 : Bool;
      _w6 : Bool;
   END_VAR
BEGIN

REGION Network 1: 调用机器人1 / Call robot 1
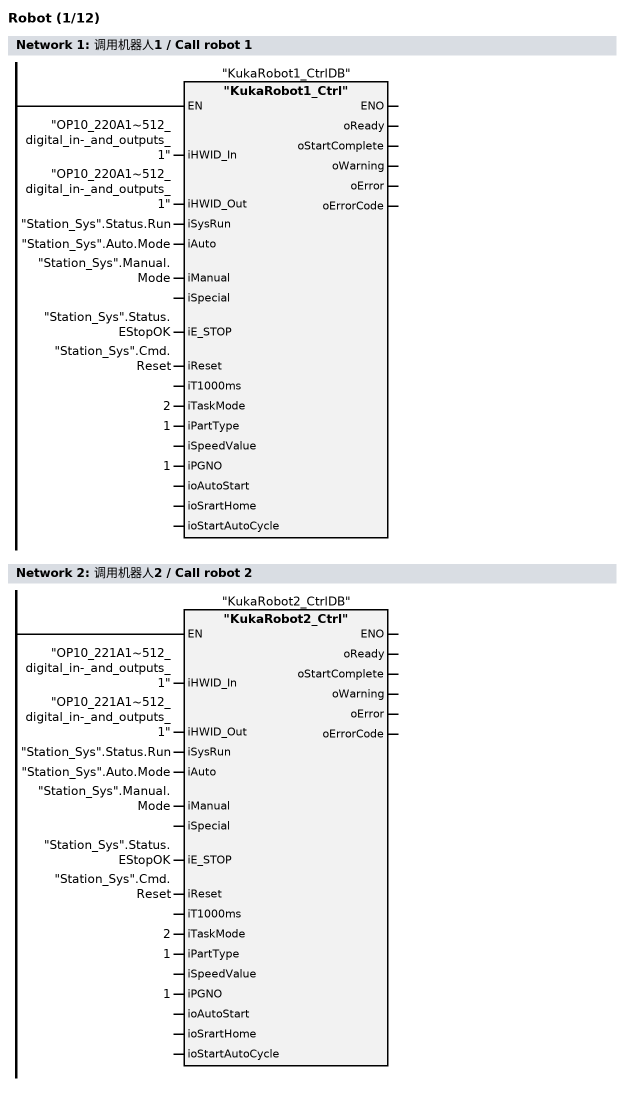
   RUNG wire#powerrail
      "KukaRobot1_CtrlDB"(iHWID_In := "OP10_220A1~512_digital_in-_and_outputs_1", iHWID_Out := "OP10_220A1~512_digital_in-_and_outputs_1", iSysRun := "Station_Sys".Status.Run, iAuto := "Station_Sys".Auto.Mode, iManual := "Station_Sys".Manual.Mode, iSpecial :=, iE_STOP := "Station_Sys".Status.EStopOK, iReset := "Station_Sys".Cmd.Reset, iT1000ms :=, iTaskMode := 2, iPartType := 1, iSpeedValue :=, iPGNO := 1, ioAutoStart :=, ioSrartHome :=, ioStartAutoCycle :=, oReady =>, oStartComplete =>, oWarning =>, oError =>, oErrorCode =>)
   END_RUNG
   // the same network as SCL:
   "KukaRobot1_CtrlDB"(iHWID_In := "OP10_220A1~512_digital_in-_and_outputs_1",   // "KukaRobot1_Ctrl"
                       iHWID_Out := "OP10_220A1~512_digital_in-_and_outputs_1",
                       iSysRun := "Station_Sys".Status.Run,
                       iAuto := "Station_Sys".Auto.Mode,
                       iManual := "Station_Sys".Manual.Mode,
                       iE_STOP := "Station_Sys".Status.EStopOK,
                       iReset := "Station_Sys".Cmd.Reset,
                       iTaskMode := 2,
                       iPartType := 1,
                       iPGNO := 1);
END_REGION

REGION Network 2: 调用机器人2 / Call robot 2
   RUNG wire#powerrail
      "KukaRobot2_CtrlDB"(iHWID_In := "OP10_221A1~512_digital_in-_and_outputs_1", iHWID_Out := "OP10_221A1~512_digital_in-_and_outputs_1", iSysRun := "Station_Sys".Status.Run, iAuto := "Station_Sys".Auto.Mode, iManual := "Station_Sys".Manual.Mode, iSpecial :=, iE_STOP := "Station_Sys".Status.EStopOK, iReset := "Station_Sys".Cmd.Reset, iT1000ms :=, iTaskMode := 2, iPartType := 1, iSpeedValue :=, iPGNO := 1, ioAutoStart :=, ioSrartHome :=, ioStartAutoCycle :=, oReady =>, oStartComplete =>, oWarning =>, oError =>, oErrorCode =>)
   END_RUNG
   // the same network as SCL:
   "KukaRobot2_CtrlDB"(iHWID_In := "OP10_221A1~512_digital_in-_and_outputs_1",   // "KukaRobot2_Ctrl"
                       iHWID_Out := "OP10_221A1~512_digital_in-_and_outputs_1",
                       iSysRun := "Station_Sys".Status.Run,
                       iAuto := "Station_Sys".Auto.Mode,
                       iManual := "Station_Sys".Manual.Mode,
                       iE_STOP := "Station_Sys".Status.EStopOK,
                       iReset := "Station_Sys".Cmd.Reset,
                       iTaskMode := 2,
                       iPartType := 1,
                       iPGNO := 1);
END_REGION

REGION Network 3: 调用机器人3 / Call robot 3
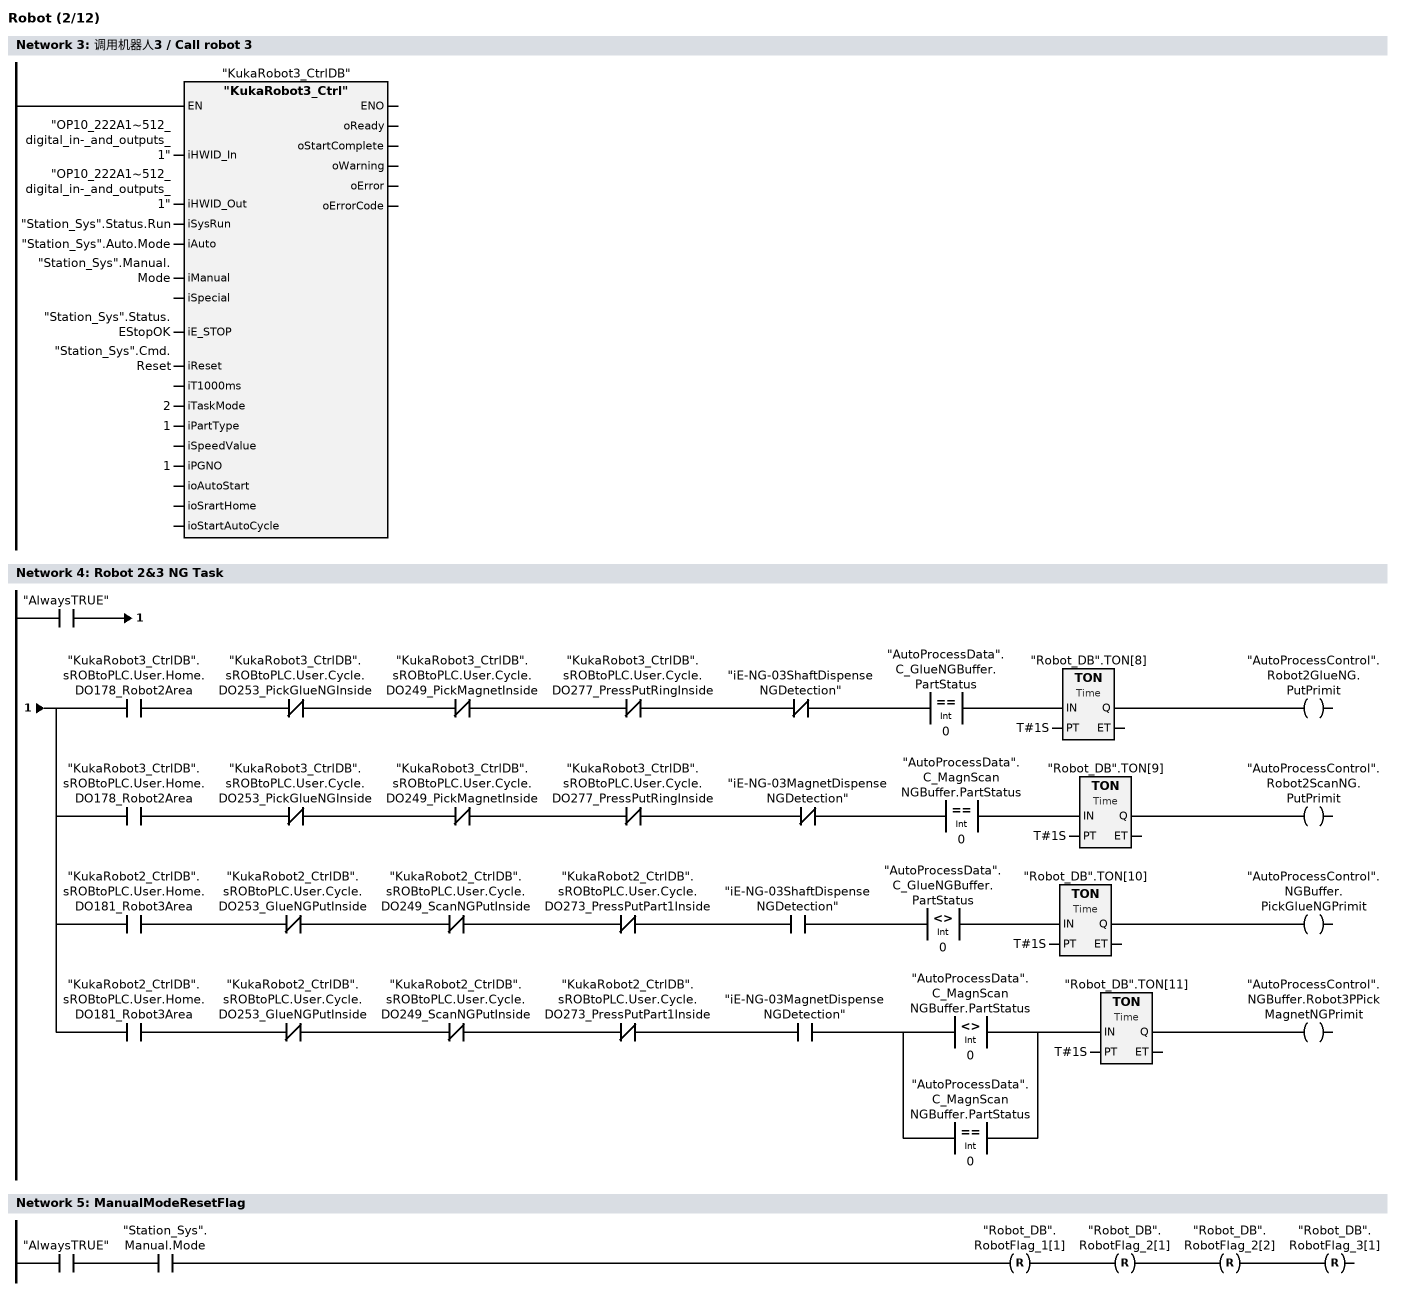
   RUNG wire#powerrail
      "KukaRobot3_CtrlDB"(iHWID_In := "OP10_222A1~512_digital_in-_and_outputs_1", iHWID_Out := "OP10_222A1~512_digital_in-_and_outputs_1", iSysRun := "Station_Sys".Status.Run, iAuto := "Station_Sys".Auto.Mode, iManual := "Station_Sys".Manual.Mode, iSpecial :=, iE_STOP := "Station_Sys".Status.EStopOK, iReset := "Station_Sys".Cmd.Reset, iT1000ms :=, iTaskMode := 2, iPartType := 1, iSpeedValue :=, iPGNO := 1, ioAutoStart :=, ioSrartHome :=, ioStartAutoCycle :=, oReady =>, oStartComplete =>, oWarning =>, oError =>, oErrorCode =>)
   END_RUNG
   // the same network as SCL:
   "KukaRobot3_CtrlDB"(iHWID_In := "OP10_222A1~512_digital_in-_and_outputs_1",   // "KukaRobot3_Ctrl"
                       iHWID_Out := "OP10_222A1~512_digital_in-_and_outputs_1",
                       iSysRun := "Station_Sys".Status.Run,
                       iAuto := "Station_Sys".Auto.Mode,
                       iManual := "Station_Sys".Manual.Mode,
                       iE_STOP := "Station_Sys".Status.EStopOK,
                       iReset := "Station_Sys".Cmd.Reset,
                       iTaskMode := 2,
                       iPartType := 1,
                       iPGNO := 1);
END_REGION

REGION Network 4: Robot 2&3 NG Task
   RUNG wire#powerrail
      Contact( "AlwaysTRUE" )
      wire#w1
      Contact( "KukaRobot3_CtrlDB".sROBtoPLC.User.Home.DO178_Robot2Area )
      I_Contact( "KukaRobot3_CtrlDB".sROBtoPLC.User.Cycle.DO253_PickGlueNGInside )
      I_Contact( "KukaRobot3_CtrlDB".sROBtoPLC.User.Cycle.DO249_PickMagnetInside )
      I_Contact( "KukaRobot3_CtrlDB".sROBtoPLC.User.Cycle.DO277_PressPutRingInside )
      I_Contact( "iE-NG-03ShaftDispenseNGDetection" )
      { S7_Templates := "SrcType := Int" } EQ_Contact(in1 := "AutoProcessData".C_GlueNGBuffer.PartStatus, in2 := 0)
      { S7_Templates := "time_type := Time" } "Robot_DB".TON[8].TON(pt := T#1S, et =>)
      Coil( "AutoProcessControl".Robot2GlueNG.PutPrimit )
   END_RUNG
   RUNG wire#w1
      Contact( "KukaRobot3_CtrlDB".sROBtoPLC.User.Home.DO178_Robot2Area )
      I_Contact( "KukaRobot3_CtrlDB".sROBtoPLC.User.Cycle.DO253_PickGlueNGInside )
      I_Contact( "KukaRobot3_CtrlDB".sROBtoPLC.User.Cycle.DO249_PickMagnetInside )
      I_Contact( "KukaRobot3_CtrlDB".sROBtoPLC.User.Cycle.DO277_PressPutRingInside )
      I_Contact( "iE-NG-03MagnetDispenseNGDetection" )
      { S7_Templates := "SrcType := Int" } EQ_Contact(in1 := "AutoProcessData".C_MagnScanNGBuffer.PartStatus, in2 := 0)
      { S7_Templates := "time_type := Time" } "Robot_DB".TON[9].TON(pt := T#1S, et =>)
      Coil( "AutoProcessControl".Robot2ScanNG.PutPrimit )
   END_RUNG
   RUNG wire#w1
      Contact( "KukaRobot2_CtrlDB".sROBtoPLC.User.Home.DO181_Robot3Area )
      I_Contact( "KukaRobot2_CtrlDB".sROBtoPLC.User.Cycle.DO253_GlueNGPutInside )
      I_Contact( "KukaRobot2_CtrlDB".sROBtoPLC.User.Cycle.DO249_ScanNGPutInside )
      I_Contact( "KukaRobot2_CtrlDB".sROBtoPLC.User.Cycle.DO273_PressPutPart1Inside )
      Contact( "iE-NG-03ShaftDispenseNGDetection" )
      { S7_Templates := "SrcType := Int" } NE_Contact(in1 := "AutoProcessData".C_GlueNGBuffer.PartStatus, in2 := 0)
      { S7_Templates := "time_type := Time" } "Robot_DB".TON[10].TON(pt := T#1S, et =>)
      Coil( "AutoProcessControl".NGBuffer.PickGlueNGPrimit )
   END_RUNG
   RUNG wire#w1
      Contact( "KukaRobot2_CtrlDB".sROBtoPLC.User.Home.DO181_Robot3Area )
      I_Contact( "KukaRobot2_CtrlDB".sROBtoPLC.User.Cycle.DO253_GlueNGPutInside )
      I_Contact( "KukaRobot2_CtrlDB".sROBtoPLC.User.Cycle.DO249_ScanNGPutInside )
      I_Contact( "KukaRobot2_CtrlDB".sROBtoPLC.User.Cycle.DO273_PressPutPart1Inside )
      Contact( "iE-NG-03MagnetDispenseNGDetection" )
      wire#w2
      { S7_Templates := "SrcType := Int" } NE_Contact(in1 := "AutoProcessData".C_MagnScanNGBuffer.PartStatus, in2 := 0)
      wire#w3
      { S7_Templates := "time_type := Time" } "Robot_DB".TON[11].TON(pt := T#1S, et =>)
      Coil( "AutoProcessControl".NGBuffer.Robot3PPickMagnetNGPrimit )
   END_RUNG
   RUNG wire#w2
      { S7_Templates := "SrcType := Int" } EQ_Contact(in1 := "AutoProcessData".C_MagnScanNGBuffer.PartStatus, in2 := 0)
   END_RUNG wire#w3
   // the same network as SCL:
   "Robot_DB".TON[8].TON(IN := "AlwaysTRUE" AND "KukaRobot3_CtrlDB".sROBtoPLC.User.Home.DO178_Robot2Area AND NOT "KukaRobot3_CtrlDB".sROBtoPLC.User.Cycle.DO253_PickGlueNGInside AND NOT "KukaRobot3_CtrlDB".sROBtoPLC.User.Cycle.DO249_PickMagnetInside AND NOT "KukaRobot3_CtrlDB".sROBtoPLC.User.Cycle.DO277_PressPutRingInside AND NOT "iE-NG-03ShaftDispenseNGDetection" AND ("AutoProcessData".C_GlueNGBuffer.PartStatus = 0),
                         PT := T#1S);
   "AutoProcessControl".Robot2GlueNG.PutPrimit := "Robot_DB".TON[8].Q;
   "Robot_DB".TON[9].TON(IN := "AlwaysTRUE" AND "KukaRobot3_CtrlDB".sROBtoPLC.User.Home.DO178_Robot2Area AND NOT "KukaRobot3_CtrlDB".sROBtoPLC.User.Cycle.DO253_PickGlueNGInside AND NOT "KukaRobot3_CtrlDB".sROBtoPLC.User.Cycle.DO249_PickMagnetInside AND NOT "KukaRobot3_CtrlDB".sROBtoPLC.User.Cycle.DO277_PressPutRingInside AND NOT "iE-NG-03MagnetDispenseNGDetection" AND ("AutoProcessData".C_MagnScanNGBuffer.PartStatus = 0),
                         PT := T#1S);
   "AutoProcessControl".Robot2ScanNG.PutPrimit := "Robot_DB".TON[9].Q;
   "Robot_DB".TON[10].TON(IN := "AlwaysTRUE" AND "KukaRobot2_CtrlDB".sROBtoPLC.User.Home.DO181_Robot3Area AND NOT "KukaRobot2_CtrlDB".sROBtoPLC.User.Cycle.DO253_GlueNGPutInside AND NOT "KukaRobot2_CtrlDB".sROBtoPLC.User.Cycle.DO249_ScanNGPutInside AND NOT "KukaRobot2_CtrlDB".sROBtoPLC.User.Cycle.DO273_PressPutPart1Inside AND "iE-NG-03ShaftDispenseNGDetection" AND ("AutoProcessData".C_GlueNGBuffer.PartStatus <> 0),
                          PT := T#1S);
   "AutoProcessControl".NGBuffer.PickGlueNGPrimit := "Robot_DB".TON[10].Q;
   "Robot_DB".TON[11].TON(IN := "AlwaysTRUE" AND "KukaRobot2_CtrlDB".sROBtoPLC.User.Home.DO181_Robot3Area AND NOT "KukaRobot2_CtrlDB".sROBtoPLC.User.Cycle.DO253_GlueNGPutInside AND NOT "KukaRobot2_CtrlDB".sROBtoPLC.User.Cycle.DO249_ScanNGPutInside AND NOT "KukaRobot2_CtrlDB".sROBtoPLC.User.Cycle.DO273_PressPutPart1Inside AND "iE-NG-03MagnetDispenseNGDetection" AND (("AutoProcessData".C_MagnScanNGBuffer.PartStatus <> 0) OR ("AutoProcessData".C_MagnScanNGBuffer.PartStatus = 0)),
                          PT := T#1S);
   "AutoProcessControl".NGBuffer.Robot3PPickMagnetNGPrimit := "Robot_DB".TON[11].Q;
END_REGION

REGION Network 5: ManualModeResetFlag
   RUNG wire#powerrail
      Contact( "AlwaysTRUE" )
      Contact( "Station_Sys".Manual.Mode )
      R_Coil( "Robot_DB".RobotFlag_1[1] )
      R_Coil( "Robot_DB".RobotFlag_2[1] )
      R_Coil( "Robot_DB".RobotFlag_2[2] )
      R_Coil( "Robot_DB".RobotFlag_3[1] )
   END_RUNG
   // the same network as SCL:
   IF "AlwaysTRUE" AND "Station_Sys".Manual.Mode THEN
       "Robot_DB".RobotFlag_1[1] := FALSE;
       "Robot_DB".RobotFlag_2[1] := FALSE;
       "Robot_DB".RobotFlag_2[2] := FALSE;
       "Robot_DB".RobotFlag_3[1] := FALSE;
   END_IF;
END_REGION

REGION Network 6 (SCL): LoadNG传感器 / Loadng sensor
   //NG1
   "KukaRobot1_CtrlDB".sPLCtoROB.User.Home.DI177_NG1_1:="Robot_DB".LoadNG_1[1] := NOT  "iE1-UnloadingShaftPressNG_5";
   "KukaRobot1_CtrlDB".sPLCtoROB.User.Home.DI178_NG1_2:="Robot_DB".LoadNG_1[2] := NOT  "iE1-UnloadingShaftPressNG_4";
   "KukaRobot1_CtrlDB".sPLCtoROB.User.Home.DI179_NG1_3:="Robot_DB".LoadNG_1[3] := NOT  "iE1-UnloadingShaftPressNG_3";
   "KukaRobot1_CtrlDB".sPLCtoROB.User.Home.DI180_NG1_4:="Robot_DB".LoadNG_1[4] := NOT  "iE1-UnloadingShaftPressNG_2";
   "KukaRobot1_CtrlDB".sPLCtoROB.User.Home.DI181_NG1_5:="Robot_DB".LoadNG_1[5] := NOT  "iE1-UnloadingShaftPressNG_1";

   //NG2
   "KukaRobot1_CtrlDB".sPLCtoROB.User.Home.DI182_NG2_1:="Robot_DB".LoadNG_2[1] := NOT  "iE1-UnloadingShaftScanNG_5";
   "KukaRobot1_CtrlDB".sPLCtoROB.User.Home.DI183_NG2_2:="Robot_DB".LoadNG_2[2] := NOT  "iE1-UnloadingShaftScanNG_4";
   "KukaRobot1_CtrlDB".sPLCtoROB.User.Home.DI184_NG2_3:="Robot_DB".LoadNG_2[3] := NOT  "iE1-UnloadingShaftScanNG_3";
   "KukaRobot1_CtrlDB".sPLCtoROB.User.Home.DI185_NG2_4:="Robot_DB".LoadNG_2[4] := NOT  "iE1-UnloadingShaftScanNG_2";
   "KukaRobot1_CtrlDB".sPLCtoROB.User.Home.DI186_NG2_5:="Robot_DB".LoadNG_2[5] := NOT  "iE1-UnloadingShaftScanNG_1";

   //NG3
   "KukaRobot1_CtrlDB".sPLCtoROB.User.Home.DI187_NG3_1:="Robot_DB".LoadNG_3[1] := NOT  "iE1-UnloadingRingScanNG_5";
   "KukaRobot1_CtrlDB".sPLCtoROB.User.Home.DI188_NG3_2:="Robot_DB".LoadNG_3[2] := NOT  "iE1-UnloadingRingScanNG_4";
   "KukaRobot1_CtrlDB".sPLCtoROB.User.Home.DI189_NG3_3:="Robot_DB".LoadNG_3[3] := NOT  "iE1-UnloadingRingScanNG_3";
   "KukaRobot1_CtrlDB".sPLCtoROB.User.Home.DI190_NG3_4:="Robot_DB".LoadNG_3[4] := NOT  "iE1-UnloadingRingScanNG_2";
   "KukaRobot1_CtrlDB".sPLCtoROB.User.Home.DI191_NG3_5:="Robot_DB".LoadNG_3[5] := NOT  "iE1-UnloadingRingScanNG_1";
END_REGION

REGION Network 7 (SCL): UnLoadNG传感器 / UnLoadNG sensor
   //NG1
   "KukaRobot3_CtrlDB".sPLCtoROB.User.Home.DI177_PressNG1_1:="Robot_DB".UnLoadNG_1[1] := NOT  "iE2-UnloadingPressNG_5";
   "KukaRobot3_CtrlDB".sPLCtoROB.User.Home.DI178_PressNG1_2:="Robot_DB".UnLoadNG_1[2] := NOT  "iE2-UnloadingPressNG_4";
   "KukaRobot3_CtrlDB".sPLCtoROB.User.Home.DI179_PressNG1_3:="Robot_DB".UnLoadNG_1[3] := NOT  "iE2-UnloadingPressNG_3";
   "KukaRobot3_CtrlDB".sPLCtoROB.User.Home.DI180_PressNG1_4:="Robot_DB".UnLoadNG_1[4] := NOT  "iE2-UnloadingPressNG_2";
   "KukaRobot3_CtrlDB".sPLCtoROB.User.Home.DI181_PressNG1_5:="Robot_DB".UnLoadNG_1[5] := NOT  "iE2-UnloadingPressNG_1";

   //NG2
   "KukaRobot3_CtrlDB".sPLCtoROB.User.Home.DI182_GlueNG2_1:="Robot_DB".UnLoadNG_2[1] := NOT  "iE2-UnloadingMagentScanNG_5";
   "KukaRobot3_CtrlDB".sPLCtoROB.User.Home.DI183_GlueNG2_2:="Robot_DB".UnLoadNG_2[2] := NOT  "iE2-UnloadingMagentScanNG_4";
   "KukaRobot3_CtrlDB".sPLCtoROB.User.Home.DI184_GlueNG2_3:="Robot_DB".UnLoadNG_2[3] := NOT  "iE2-UnloadingMagentScanNG_3";
   "KukaRobot3_CtrlDB".sPLCtoROB.User.Home.DI185_GlueNG2_4:="Robot_DB".UnLoadNG_2[4] := NOT  "iE2-UnloadingMagentScanNG_2";
   "KukaRobot3_CtrlDB".sPLCtoROB.User.Home.DI186_GlueNG2_5:="Robot_DB".UnLoadNG_2[5] := NOT  "iE2-UnloadingMagentScanNG_1";

   //NG3
   "KukaRobot3_CtrlDB".sPLCtoROB.User.Home.DI187_ScanNG3_1:="Robot_DB".UnLoadNG_3[1] := NOT  "iE2-UnloadingRingScanNG_5";
   "KukaRobot3_CtrlDB".sPLCtoROB.User.Home.DI188_ScanNG3_2:="Robot_DB".UnLoadNG_3[2] := NOT  "iE2-UnloadingRingScanNG_4";
   "KukaRobot3_CtrlDB".sPLCtoROB.User.Home.DI189_ScanNG3_3:="Robot_DB".UnLoadNG_3[3] := NOT  "iE2-UnloadingRingScanNG_3";
   "KukaRobot3_CtrlDB".sPLCtoROB.User.Home.DI190_ScanNG3_4:="Robot_DB".UnLoadNG_3[4] := NOT  "iE2-UnloadingRingScanNG_2";
   "KukaRobot3_CtrlDB".sPLCtoROB.User.Home.DI191_ScanNG3_5:="Robot_DB".UnLoadNG_3[5] := NOT  "iE2-UnloadingRingScanNG_1";
END_REGION

REGION Network 8: RobotGripControl
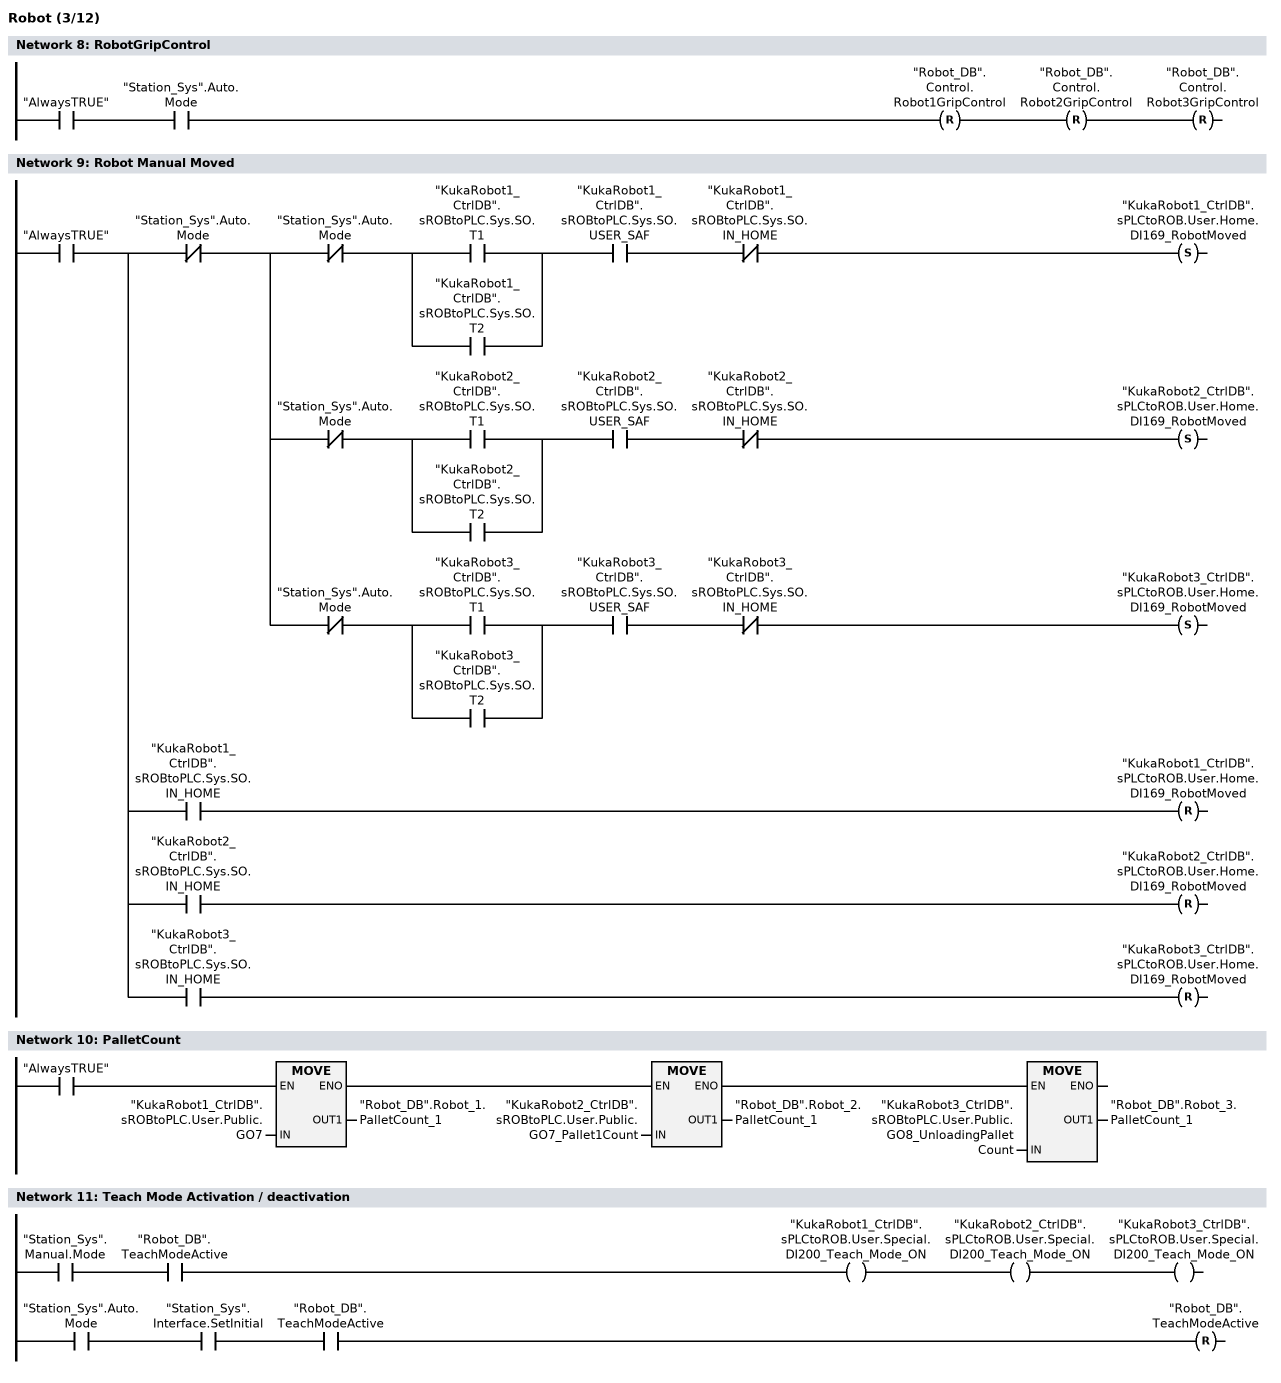
   RUNG wire#powerrail
      Contact( "AlwaysTRUE" )
      Contact( "Station_Sys".Auto.Mode )
      R_Coil( "Robot_DB".Control.Robot1GripControl )
      R_Coil( "Robot_DB".Control.Robot2GripControl )
      R_Coil( "Robot_DB".Control.Robot3GripControl )
   END_RUNG
   // the same network as SCL:
   IF "AlwaysTRUE" AND "Station_Sys".Auto.Mode THEN
       "Robot_DB".Control.Robot1GripControl := FALSE;
       "Robot_DB".Control.Robot2GripControl := FALSE;
       "Robot_DB".Control.Robot3GripControl := FALSE;
   END_IF;
END_REGION

REGION Network 9: Robot Manual Moved
   RUNG wire#powerrail
      Contact( "AlwaysTRUE" )
      wire#w1
      I_Contact( "Station_Sys".Auto.Mode )
      wire#w2
      I_Contact( "Station_Sys".Auto.Mode )
      wire#w3
      Contact( "KukaRobot1_CtrlDB".sROBtoPLC.Sys.SO.T1 )
      wire#w4
      Contact( "KukaRobot1_CtrlDB".sROBtoPLC.Sys.SO.USER_SAF )
      I_Contact( "KukaRobot1_CtrlDB".sROBtoPLC.Sys.SO.IN_HOME )
      S_Coil( "KukaRobot1_CtrlDB".sPLCtoROB.User.Home.DI169_RobotMoved )
   END_RUNG
   RUNG wire#w3
      Contact( "KukaRobot1_CtrlDB".sROBtoPLC.Sys.SO.T2 )
   END_RUNG wire#w4
   RUNG wire#w2
      I_Contact( "Station_Sys".Auto.Mode )
      wire#w5
      Contact( "KukaRobot2_CtrlDB".sROBtoPLC.Sys.SO.T1 )
      wire#w6
      Contact( "KukaRobot2_CtrlDB".sROBtoPLC.Sys.SO.USER_SAF )
      I_Contact( "KukaRobot2_CtrlDB".sROBtoPLC.Sys.SO.IN_HOME )
      S_Coil( "KukaRobot2_CtrlDB".sPLCtoROB.User.Home.DI169_RobotMoved )
   END_RUNG
   RUNG wire#w5
      Contact( "KukaRobot2_CtrlDB".sROBtoPLC.Sys.SO.T2 )
   END_RUNG wire#w6
   RUNG wire#w2
      I_Contact( "Station_Sys".Auto.Mode )
      wire#w7
      Contact( "KukaRobot3_CtrlDB".sROBtoPLC.Sys.SO.T1 )
      wire#w8
      Contact( "KukaRobot3_CtrlDB".sROBtoPLC.Sys.SO.USER_SAF )
      I_Contact( "KukaRobot3_CtrlDB".sROBtoPLC.Sys.SO.IN_HOME )
      S_Coil( "KukaRobot3_CtrlDB".sPLCtoROB.User.Home.DI169_RobotMoved )
   END_RUNG
   RUNG wire#w7
      Contact( "KukaRobot3_CtrlDB".sROBtoPLC.Sys.SO.T2 )
   END_RUNG wire#w8
   RUNG wire#w1
      Contact( "KukaRobot1_CtrlDB".sROBtoPLC.Sys.SO.IN_HOME )
      R_Coil( "KukaRobot1_CtrlDB".sPLCtoROB.User.Home.DI169_RobotMoved )
   END_RUNG
   RUNG wire#w1
      Contact( "KukaRobot2_CtrlDB".sROBtoPLC.Sys.SO.IN_HOME )
      R_Coil( "KukaRobot2_CtrlDB".sPLCtoROB.User.Home.DI169_RobotMoved )
   END_RUNG
   RUNG wire#w1
      Contact( "KukaRobot3_CtrlDB".sROBtoPLC.Sys.SO.IN_HOME )
      R_Coil( "KukaRobot3_CtrlDB".sPLCtoROB.User.Home.DI169_RobotMoved )
   END_RUNG
   // the same network as SCL:
   #_w1 := "AlwaysTRUE" AND NOT "Station_Sys".Auto.Mode;
   IF #_w1 AND NOT "Station_Sys".Auto.Mode AND ("KukaRobot1_CtrlDB".sROBtoPLC.Sys.SO.T1 OR "KukaRobot1_CtrlDB".sROBtoPLC.Sys.SO.T2) AND "KukaRobot1_CtrlDB".sROBtoPLC.Sys.SO.USER_SAF AND NOT "KukaRobot1_CtrlDB".sROBtoPLC.Sys.SO.IN_HOME THEN
       "KukaRobot1_CtrlDB".sPLCtoROB.User.Home.DI169_RobotMoved := TRUE;
   END_IF;
   IF #_w1 AND NOT "Station_Sys".Auto.Mode AND ("KukaRobot2_CtrlDB".sROBtoPLC.Sys.SO.T1 OR "KukaRobot2_CtrlDB".sROBtoPLC.Sys.SO.T2) AND "KukaRobot2_CtrlDB".sROBtoPLC.Sys.SO.USER_SAF AND NOT "KukaRobot2_CtrlDB".sROBtoPLC.Sys.SO.IN_HOME THEN
       "KukaRobot2_CtrlDB".sPLCtoROB.User.Home.DI169_RobotMoved := TRUE;
   END_IF;
   IF #_w1 AND NOT "Station_Sys".Auto.Mode AND ("KukaRobot3_CtrlDB".sROBtoPLC.Sys.SO.T1 OR "KukaRobot3_CtrlDB".sROBtoPLC.Sys.SO.T2) AND "KukaRobot3_CtrlDB".sROBtoPLC.Sys.SO.USER_SAF AND NOT "KukaRobot3_CtrlDB".sROBtoPLC.Sys.SO.IN_HOME THEN
       "KukaRobot3_CtrlDB".sPLCtoROB.User.Home.DI169_RobotMoved := TRUE;
   END_IF;
   IF "AlwaysTRUE" AND "KukaRobot1_CtrlDB".sROBtoPLC.Sys.SO.IN_HOME THEN
       "KukaRobot1_CtrlDB".sPLCtoROB.User.Home.DI169_RobotMoved := FALSE;
   END_IF;
   IF "AlwaysTRUE" AND "KukaRobot2_CtrlDB".sROBtoPLC.Sys.SO.IN_HOME THEN
       "KukaRobot2_CtrlDB".sPLCtoROB.User.Home.DI169_RobotMoved := FALSE;
   END_IF;
   IF "AlwaysTRUE" AND "KukaRobot3_CtrlDB".sROBtoPLC.Sys.SO.IN_HOME THEN
       "KukaRobot3_CtrlDB".sPLCtoROB.User.Home.DI169_RobotMoved := FALSE;
   END_IF;
END_REGION

REGION Network 10: PalletCount
   RUNG wire#powerrail
      Contact( "AlwaysTRUE" )
      Move(in := "KukaRobot1_CtrlDB".sROBtoPLC.User.Public.GO7, out1 => "Robot_DB".Robot_1.PalletCount_1)
      Move(in := "KukaRobot2_CtrlDB".sROBtoPLC.User.Public.GO7_Pallet1Count, out1 => "Robot_DB".Robot_2.PalletCount_1)
      Move(in := "KukaRobot3_CtrlDB".sROBtoPLC.User.Public.GO8_UnloadingPalletCount, out1 => "Robot_DB".Robot_3.PalletCount_1)
   END_RUNG
   // the same network as SCL:
   IF "AlwaysTRUE" THEN
       "Robot_DB".Robot_1.PalletCount_1 := "KukaRobot1_CtrlDB".sROBtoPLC.User.Public.GO7;
       "Robot_DB".Robot_2.PalletCount_1 := "KukaRobot2_CtrlDB".sROBtoPLC.User.Public.GO7_Pallet1Count;
       "Robot_DB".Robot_3.PalletCount_1 := "KukaRobot3_CtrlDB".sROBtoPLC.User.Public.GO8_UnloadingPalletCount;
   END_IF;
END_REGION

REGION Network 11: Teach Mode Activation / deactivation
   RUNG wire#powerrail
      Contact( "Station_Sys".Manual.Mode )
      Contact( "Robot_DB".TeachModeActive )
      Coil( "KukaRobot1_CtrlDB".sPLCtoROB.User.Special.DI200_Teach_Mode_ON )
      Coil( "KukaRobot2_CtrlDB".sPLCtoROB.User.Special.DI200_Teach_Mode_ON )
      Coil( "KukaRobot3_CtrlDB".sPLCtoROB.User.Special.DI200_Teach_Mode_ON )
   END_RUNG
   RUNG wire#powerrail
      Contact( "Station_Sys".Auto.Mode )
      Contact( "Station_Sys".Interface.SetInitial )
      Contact( "Robot_DB".TeachModeActive )
      R_Coil( "Robot_DB".TeachModeActive )
   END_RUNG
   // the same network as SCL:
   "KukaRobot1_CtrlDB".sPLCtoROB.User.Special.DI200_Teach_Mode_ON := "Station_Sys".Manual.Mode AND "Robot_DB".TeachModeActive;
   "KukaRobot2_CtrlDB".sPLCtoROB.User.Special.DI200_Teach_Mode_ON := "KukaRobot1_CtrlDB".sPLCtoROB.User.Special.DI200_Teach_Mode_ON;
   "KukaRobot3_CtrlDB".sPLCtoROB.User.Special.DI200_Teach_Mode_ON := "KukaRobot1_CtrlDB".sPLCtoROB.User.Special.DI200_Teach_Mode_ON;
   IF "Station_Sys".Auto.Mode AND "Station_Sys".Interface.SetInitial AND "Robot_DB".TeachModeActive THEN
       "Robot_DB".TeachModeActive := FALSE;
   END_IF;
END_REGION

REGION Network 13: ----------------------------------------- Robot_1 -------------------------------------
END_REGION

REGION Network 14: CodeCompare
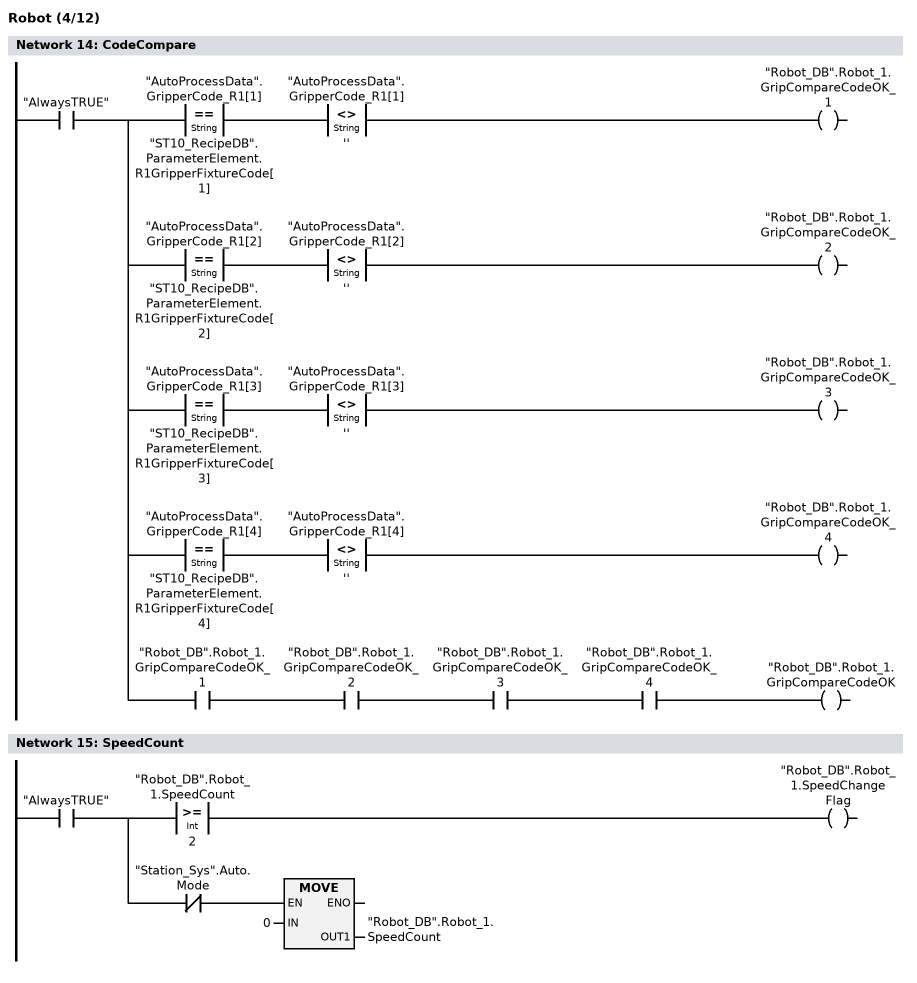
   RUNG wire#powerrail
      Contact( "AlwaysTRUE" )
      wire#w1
      { S7_Templates := "SrcType := String" } EQ_Contact(in1 := "AutoProcessData".GripperCode_R1[1], in2 := "ST10_RecipeDB".ParameterElement.R1GripperFixtureCode[1])
      { S7_Templates := "SrcType := String" } NE_Contact(in1 := "AutoProcessData".GripperCode_R1[1], in2 := '')
      Coil( "Robot_DB".Robot_1.GripCompareCodeOK_1 )
   END_RUNG
   RUNG wire#w1
      { S7_Templates := "SrcType := String" } EQ_Contact(in1 := "AutoProcessData".GripperCode_R1[2], in2 := "ST10_RecipeDB".ParameterElement.R1GripperFixtureCode[2])
      { S7_Templates := "SrcType := String" } NE_Contact(in1 := "AutoProcessData".GripperCode_R1[2], in2 := '')
      Coil( "Robot_DB".Robot_1.GripCompareCodeOK_2 )
   END_RUNG
   RUNG wire#w1
      { S7_Templates := "SrcType := String" } EQ_Contact(in1 := "AutoProcessData".GripperCode_R1[3], in2 := "ST10_RecipeDB".ParameterElement.R1GripperFixtureCode[3])
      { S7_Templates := "SrcType := String" } NE_Contact(in1 := "AutoProcessData".GripperCode_R1[3], in2 := '')
      Coil( "Robot_DB".Robot_1.GripCompareCodeOK_3 )
   END_RUNG
   RUNG wire#w1
      { S7_Templates := "SrcType := String" } EQ_Contact(in1 := "AutoProcessData".GripperCode_R1[4], in2 := "ST10_RecipeDB".ParameterElement.R1GripperFixtureCode[4])
      { S7_Templates := "SrcType := String" } NE_Contact(in1 := "AutoProcessData".GripperCode_R1[4], in2 := '')
      Coil( "Robot_DB".Robot_1.GripCompareCodeOK_4 )
   END_RUNG
   RUNG wire#w1
      Contact( "Robot_DB".Robot_1.GripCompareCodeOK_1 )
      Contact( "Robot_DB".Robot_1.GripCompareCodeOK_2 )
      Contact( "Robot_DB".Robot_1.GripCompareCodeOK_3 )
      Contact( "Robot_DB".Robot_1.GripCompareCodeOK_4 )
      Coil( "Robot_DB".Robot_1.GripCompareCodeOK )
   END_RUNG
   // the same network as SCL:
   "Robot_DB".Robot_1.GripCompareCodeOK_1 := "AlwaysTRUE" AND ("AutoProcessData".GripperCode_R1[1] = "ST10_RecipeDB".ParameterElement.R1GripperFixtureCode[1]) AND ("AutoProcessData".GripperCode_R1[1] <> '');
   "Robot_DB".Robot_1.GripCompareCodeOK_2 := "AlwaysTRUE" AND ("AutoProcessData".GripperCode_R1[2] = "ST10_RecipeDB".ParameterElement.R1GripperFixtureCode[2]) AND ("AutoProcessData".GripperCode_R1[2] <> '');
   "Robot_DB".Robot_1.GripCompareCodeOK_3 := "AlwaysTRUE" AND ("AutoProcessData".GripperCode_R1[3] = "ST10_RecipeDB".ParameterElement.R1GripperFixtureCode[3]) AND ("AutoProcessData".GripperCode_R1[3] <> '');
   "Robot_DB".Robot_1.GripCompareCodeOK_4 := "AlwaysTRUE" AND ("AutoProcessData".GripperCode_R1[4] = "ST10_RecipeDB".ParameterElement.R1GripperFixtureCode[4]) AND ("AutoProcessData".GripperCode_R1[4] <> '');
   "Robot_DB".Robot_1.GripCompareCodeOK := "AlwaysTRUE" AND "Robot_DB".Robot_1.GripCompareCodeOK_1 AND "Robot_DB".Robot_1.GripCompareCodeOK_2 AND "Robot_DB".Robot_1.GripCompareCodeOK_3 AND "Robot_DB".Robot_1.GripCompareCodeOK_4;
END_REGION

REGION Network 15: SpeedCount
   RUNG wire#powerrail
      Contact( "AlwaysTRUE" )
      wire#w1
      { S7_Templates := "SrcType := Int" } GE_Contact(in1 := "Robot_DB".Robot_1.SpeedCount, in2 := 2)
      Coil( "Robot_DB".Robot_1.SpeedChangeFlag )
   END_RUNG
   RUNG wire#w1
      I_Contact( "Station_Sys".Auto.Mode )
      Move(in := 0, out1 => "Robot_DB".Robot_1.SpeedCount)
   END_RUNG
   // the same network as SCL:
   "Robot_DB".Robot_1.SpeedChangeFlag := "AlwaysTRUE" AND ("Robot_DB".Robot_1.SpeedCount >= 2);
   IF "AlwaysTRUE" AND NOT "Station_Sys".Auto.Mode THEN "Robot_DB".Robot_1.SpeedCount := 0; END_IF;
END_REGION

REGION Network 16: Robot1Speed Interlock
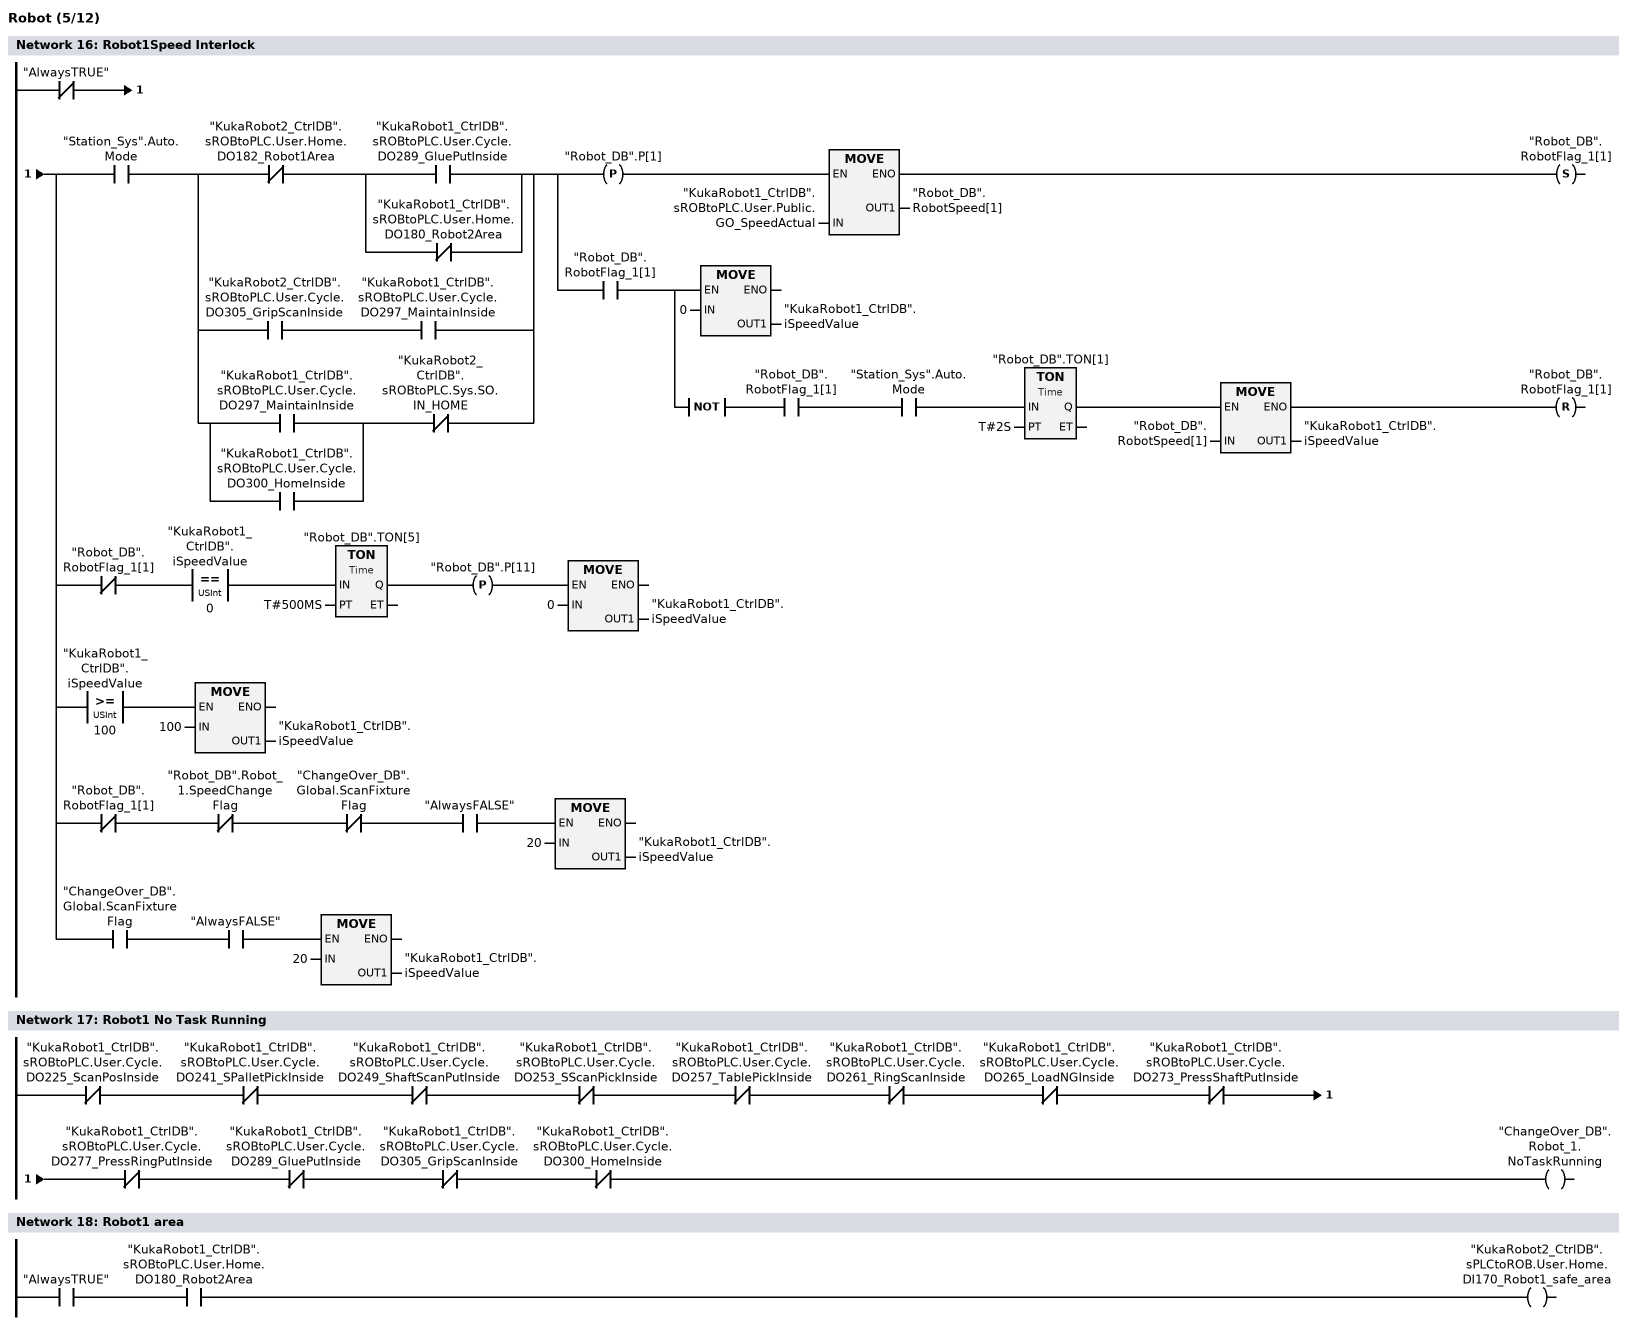
   RUNG wire#powerrail
      I_Contact( "AlwaysTRUE" )
      wire#w1
      Contact( "Station_Sys".Auto.Mode )
      wire#w2
      I_Contact( "KukaRobot2_CtrlDB".sROBtoPLC.User.Home.DO182_Robot1Area )
      wire#w3
      Contact( "KukaRobot1_CtrlDB".sROBtoPLC.User.Cycle.DO289_GluePutInside )
      wire#w4
      P_Trig( "Robot_DB".P[1] )
      Move(in := "KukaRobot1_CtrlDB".sROBtoPLC.User.Public.GO_SpeedActual, out1 => "Robot_DB".RobotSpeed[1])
      S_Coil( "Robot_DB".RobotFlag_1[1] )
   END_RUNG
   RUNG wire#w3
      I_Contact( "KukaRobot1_CtrlDB".sROBtoPLC.User.Home.DO180_Robot2Area )
   END_RUNG wire#w4
   RUNG wire#w2
      Contact( "KukaRobot2_CtrlDB".sROBtoPLC.User.Cycle.DO305_GripScanInside )
      Contact( "KukaRobot1_CtrlDB".sROBtoPLC.User.Cycle.DO297_MaintainInside )
   END_RUNG wire#w4
   RUNG wire#w2
      Contact( "KukaRobot1_CtrlDB".sROBtoPLC.User.Cycle.DO297_MaintainInside )
      wire#w5
      I_Contact( "KukaRobot2_CtrlDB".sROBtoPLC.Sys.SO.IN_HOME )
   END_RUNG wire#w4
   RUNG wire#w2
      Contact( "KukaRobot1_CtrlDB".sROBtoPLC.User.Cycle.DO300_HomeInside )
   END_RUNG wire#w5
   RUNG wire#w4
      Contact( "Robot_DB".RobotFlag_1[1] )
      wire#w6
      Move(in := 0, out1 => "KukaRobot1_CtrlDB".iSpeedValue)
   END_RUNG
   RUNG wire#w6
      Not()
      Contact( "Robot_DB".RobotFlag_1[1] )
      Contact( "Station_Sys".Auto.Mode )
      { S7_Templates := "time_type := Time" } "Robot_DB".TON[1].TON(pt := T#2S, et =>)
      Move(in := "Robot_DB".RobotSpeed[1], out1 => "KukaRobot1_CtrlDB".iSpeedValue)
      R_Coil( "Robot_DB".RobotFlag_1[1] )
   END_RUNG
   RUNG wire#w1
      I_Contact( "Robot_DB".RobotFlag_1[1] )
      { S7_Templates := "SrcType := USInt" } EQ_Contact(in1 := "KukaRobot1_CtrlDB".iSpeedValue, in2 := 0)
      { S7_Templates := "time_type := Time" } "Robot_DB".TON[5].TON(pt := T#500MS, et =>)
      P_Trig( "Robot_DB".P[11] )
      Move(in := 0, out1 => "KukaRobot1_CtrlDB".iSpeedValue)
   END_RUNG
   RUNG wire#w1
      { S7_Templates := "SrcType := USInt" } GE_Contact(in1 := "KukaRobot1_CtrlDB".iSpeedValue, in2 := 100)
      Move(in := 100, out1 => "KukaRobot1_CtrlDB".iSpeedValue)
   END_RUNG
   RUNG wire#w1
      I_Contact( "Robot_DB".RobotFlag_1[1] )
      I_Contact( "Robot_DB".Robot_1.SpeedChangeFlag )
      I_Contact( "ChangeOver_DB".Global.ScanFixtureFlag )
      Contact( "AlwaysFALSE" )
      Move(in := 20, out1 => "KukaRobot1_CtrlDB".iSpeedValue)
   END_RUNG
   RUNG wire#w1
      Contact( "ChangeOver_DB".Global.ScanFixtureFlag )
      Contact( "AlwaysFALSE" )
      Move(in := 20, out1 => "KukaRobot1_CtrlDB".iSpeedValue)
   END_RUNG
   // the same network as SCL:
   #_w1 := NOT "AlwaysTRUE" AND "Station_Sys".Auto.Mode AND ((NOT "KukaRobot2_CtrlDB".sROBtoPLC.User.Home.DO182_Robot1Area AND ("KukaRobot1_CtrlDB".sROBtoPLC.User.Cycle.DO289_GluePutInside OR NOT "KukaRobot1_CtrlDB".sROBtoPLC.User.Home.DO180_Robot2Area)) OR ("KukaRobot2_CtrlDB".sROBtoPLC.User.Cycle.DO305_GripScanInside AND "KukaRobot1_CtrlDB".sROBtoPLC.User.Cycle.DO297_MaintainInside) OR (("KukaRobot1_CtrlDB".sROBtoPLC.User.Cycle.DO297_MaintainInside OR "KukaRobot1_CtrlDB".sROBtoPLC.User.Cycle.DO300_HomeInside) AND NOT "KukaRobot2_CtrlDB".sROBtoPLC.Sys.SO.IN_HOME));
   #_w2 := #_w1 AND NOT "Robot_DB".P[1];   // rising edge
   "Robot_DB".P[1] := #_w1;
   IF #_w2 THEN
       "Robot_DB".RobotSpeed[1] := "KukaRobot1_CtrlDB".sROBtoPLC.User.Public.GO_SpeedActual;
       "Robot_DB".RobotFlag_1[1] := TRUE;
   END_IF;
   #_w3 := #_w1 AND "Robot_DB".RobotFlag_1[1];
   IF #_w3 THEN "KukaRobot1_CtrlDB".iSpeedValue := 0; END_IF;
   "Robot_DB".TON[1].TON(IN := NOT #_w3 AND "Robot_DB".RobotFlag_1[1] AND "Station_Sys".Auto.Mode, PT := T#2S);
   IF "Robot_DB".TON[1].Q THEN
       "KukaRobot1_CtrlDB".iSpeedValue := "Robot_DB".RobotSpeed[1];
       "Robot_DB".RobotFlag_1[1] := FALSE;
   END_IF;
   "Robot_DB".TON[5].TON(IN := NOT "AlwaysTRUE" AND NOT "Robot_DB".RobotFlag_1[1] AND ("KukaRobot1_CtrlDB".iSpeedValue = 0),
                         PT := T#500MS);
   #_w4 := "Robot_DB".TON[5].Q AND NOT "Robot_DB".P[11];   // rising edge
   "Robot_DB".P[11] := "Robot_DB".TON[5].Q;
   IF #_w4 THEN "KukaRobot1_CtrlDB".iSpeedValue := 0; END_IF;
   IF NOT "AlwaysTRUE" AND ("KukaRobot1_CtrlDB".iSpeedValue >= 100) THEN
       "KukaRobot1_CtrlDB".iSpeedValue := 100;
   END_IF;
   IF NOT "AlwaysTRUE" AND NOT "Robot_DB".RobotFlag_1[1] AND NOT "Robot_DB".Robot_1.SpeedChangeFlag AND NOT "ChangeOver_DB".Global.ScanFixtureFlag AND "AlwaysFALSE" THEN
       "KukaRobot1_CtrlDB".iSpeedValue := 20;
   END_IF;
   IF NOT "AlwaysTRUE" AND "ChangeOver_DB".Global.ScanFixtureFlag AND "AlwaysFALSE" THEN
       "KukaRobot1_CtrlDB".iSpeedValue := 20;
   END_IF;
END_REGION

REGION Network 17: Robot1 No Task Running
   RUNG wire#powerrail
      I_Contact( "KukaRobot1_CtrlDB".sROBtoPLC.User.Cycle.DO225_ScanPosInside )
      I_Contact( "KukaRobot1_CtrlDB".sROBtoPLC.User.Cycle.DO241_SPalletPickInside )
      I_Contact( "KukaRobot1_CtrlDB".sROBtoPLC.User.Cycle.DO249_ShaftScanPutInside )
      I_Contact( "KukaRobot1_CtrlDB".sROBtoPLC.User.Cycle.DO253_SScanPickInside )
      I_Contact( "KukaRobot1_CtrlDB".sROBtoPLC.User.Cycle.DO257_TablePickInside )
      I_Contact( "KukaRobot1_CtrlDB".sROBtoPLC.User.Cycle.DO261_RingScanInside )
      I_Contact( "KukaRobot1_CtrlDB".sROBtoPLC.User.Cycle.DO265_LoadNGInside )
      I_Contact( "KukaRobot1_CtrlDB".sROBtoPLC.User.Cycle.DO273_PressShaftPutInside )
      I_Contact( "KukaRobot1_CtrlDB".sROBtoPLC.User.Cycle.DO277_PressRingPutInside )
      I_Contact( "KukaRobot1_CtrlDB".sROBtoPLC.User.Cycle.DO289_GluePutInside )
      I_Contact( "KukaRobot1_CtrlDB".sROBtoPLC.User.Cycle.DO305_GripScanInside )
      I_Contact( "KukaRobot1_CtrlDB".sROBtoPLC.User.Cycle.DO300_HomeInside )
      Coil( "ChangeOver_DB".Robot_1.NoTaskRunning )
   END_RUNG
   // the same network as SCL:
   "ChangeOver_DB".Robot_1.NoTaskRunning := NOT "KukaRobot1_CtrlDB".sROBtoPLC.User.Cycle.DO225_ScanPosInside AND NOT "KukaRobot1_CtrlDB".sROBtoPLC.User.Cycle.DO241_SPalletPickInside AND NOT "KukaRobot1_CtrlDB".sROBtoPLC.User.Cycle.DO249_ShaftScanPutInside AND NOT "KukaRobot1_CtrlDB".sROBtoPLC.User.Cycle.DO253_SScanPickInside AND NOT "KukaRobot1_CtrlDB".sROBtoPLC.User.Cycle.DO257_TablePickInside AND NOT "KukaRobot1_CtrlDB".sROBtoPLC.User.Cycle.DO261_RingScanInside AND NOT "KukaRobot1_CtrlDB".sROBtoPLC.User.Cycle.DO265_LoadNGInside AND NOT "KukaRobot1_CtrlDB".sROBtoPLC.User.Cycle.DO273_PressShaftPutInside AND NOT "KukaRobot1_CtrlDB".sROBtoPLC.User.Cycle.DO277_PressRingPutInside AND NOT "KukaRobot1_CtrlDB".sROBtoPLC.User.Cycle.DO289_GluePutInside AND NOT "KukaRobot1_CtrlDB".sROBtoPLC.User.Cycle.DO305_GripScanInside AND NOT "KukaRobot1_CtrlDB".sROBtoPLC.User.Cycle.DO300_HomeInside;
END_REGION

REGION Network 18: Robot1 area
   RUNG wire#powerrail
      Contact( "AlwaysTRUE" )
      Contact( "KukaRobot1_CtrlDB".sROBtoPLC.User.Home.DO180_Robot2Area )
      Coil( "KukaRobot2_CtrlDB".sPLCtoROB.User.Home.DI170_Robot1_safe_area )
   END_RUNG
   // the same network as SCL:
   "KukaRobot2_CtrlDB".sPLCtoROB.User.Home.DI170_Robot1_safe_area := "AlwaysTRUE" AND "KukaRobot1_CtrlDB".sROBtoPLC.User.Home.DO180_Robot2Area;
END_REGION

REGION Network 19: MasteringTest_Req & BrakeTest_Req
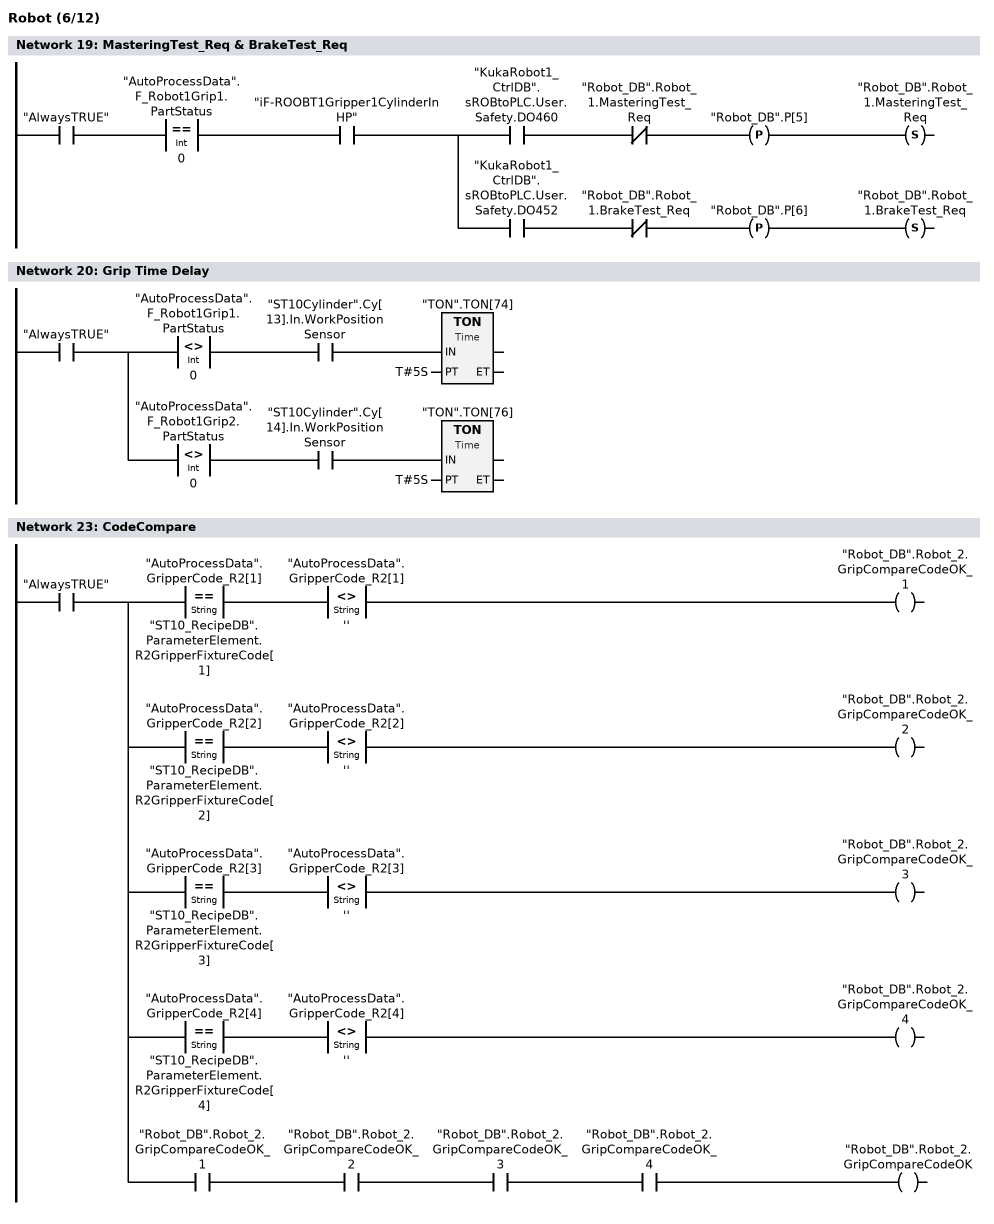
   RUNG wire#powerrail
      Contact( "AlwaysTRUE" )
      { S7_Templates := "SrcType := Int" } EQ_Contact(in1 := "AutoProcessData".F_Robot1Grip1.PartStatus, in2 := 0)
      Contact( "iF-ROOBT1Gripper1CylinderInHP" )
      wire#w1
      Contact( "KukaRobot1_CtrlDB".sROBtoPLC.User.Safety.DO460 )
      I_Contact( "Robot_DB".Robot_1.MasteringTest_Req )
      P_Trig( "Robot_DB".P[5] )
      S_Coil( "Robot_DB".Robot_1.MasteringTest_Req )
   END_RUNG
   RUNG wire#w1
      Contact( "KukaRobot1_CtrlDB".sROBtoPLC.User.Safety.DO452 )
      I_Contact( "Robot_DB".Robot_1.BrakeTest_Req )
      P_Trig( "Robot_DB".P[6] )
      S_Coil( "Robot_DB".Robot_1.BrakeTest_Req )
   END_RUNG
   // the same network as SCL:
   #_w1 := "AlwaysTRUE" AND ("AutoProcessData".F_Robot1Grip1.PartStatus = 0) AND "iF-ROOBT1Gripper1CylinderInHP";
   #_w2 := #_w1 AND "KukaRobot1_CtrlDB".sROBtoPLC.User.Safety.DO460 AND NOT "Robot_DB".Robot_1.MasteringTest_Req;
   #_w3 := #_w2 AND NOT "Robot_DB".P[5];   // rising edge
   "Robot_DB".P[5] := #_w2;
   IF #_w3 THEN "Robot_DB".Robot_1.MasteringTest_Req := TRUE; END_IF;
   #_w4 := #_w1 AND "KukaRobot1_CtrlDB".sROBtoPLC.User.Safety.DO452 AND NOT "Robot_DB".Robot_1.BrakeTest_Req;
   #_w5 := #_w4 AND NOT "Robot_DB".P[6];   // rising edge
   "Robot_DB".P[6] := #_w4;
   IF #_w5 THEN "Robot_DB".Robot_1.BrakeTest_Req := TRUE; END_IF;
END_REGION

REGION Network 20: Grip Time Delay
   RUNG wire#powerrail
      Contact( "AlwaysTRUE" )
      wire#w1
      { S7_Templates := "SrcType := Int" } NE_Contact(in1 := "AutoProcessData".F_Robot1Grip1.PartStatus, in2 := 0)
      Contact( "ST10Cylinder".Cy[13].In.WorkPositionSensor )
      { S7_Templates := "time_type := Time" } "TON".TON[74].TON(pt := T#5S, et =>)
   END_RUNG
   RUNG wire#w1
      { S7_Templates := "SrcType := Int" } NE_Contact(in1 := "AutoProcessData".F_Robot1Grip2.PartStatus, in2 := 0)
      Contact( "ST10Cylinder".Cy[14].In.WorkPositionSensor )
      { S7_Templates := "time_type := Time" } "TON".TON[76].TON(pt := T#5S, et =>)
   END_RUNG
   // the same network as SCL:
   "TON".TON[74].TON(IN := "AlwaysTRUE" AND ("AutoProcessData".F_Robot1Grip1.PartStatus <> 0) AND "ST10Cylinder".Cy[13].In.WorkPositionSensor,
                     PT := T#5S);
   "TON".TON[76].TON(IN := "AlwaysTRUE" AND ("AutoProcessData".F_Robot1Grip2.PartStatus <> 0) AND "ST10Cylinder".Cy[14].In.WorkPositionSensor,
                     PT := T#5S);
END_REGION

REGION Network 22: ----------------------------------------- Robot_2 -------------------------------------
END_REGION

REGION Network 23: CodeCompare
   RUNG wire#powerrail
      Contact( "AlwaysTRUE" )
      wire#w1
      { S7_Templates := "SrcType := String" } EQ_Contact(in1 := "AutoProcessData".GripperCode_R2[1], in2 := "ST10_RecipeDB".ParameterElement.R2GripperFixtureCode[1])
      { S7_Templates := "SrcType := String" } NE_Contact(in1 := "AutoProcessData".GripperCode_R2[1], in2 := '')
      Coil( "Robot_DB".Robot_2.GripCompareCodeOK_1 )
   END_RUNG
   RUNG wire#w1
      { S7_Templates := "SrcType := String" } EQ_Contact(in1 := "AutoProcessData".GripperCode_R2[2], in2 := "ST10_RecipeDB".ParameterElement.R2GripperFixtureCode[2])
      { S7_Templates := "SrcType := String" } NE_Contact(in1 := "AutoProcessData".GripperCode_R2[2], in2 := '')
      Coil( "Robot_DB".Robot_2.GripCompareCodeOK_2 )
   END_RUNG
   RUNG wire#w1
      { S7_Templates := "SrcType := String" } EQ_Contact(in1 := "AutoProcessData".GripperCode_R2[3], in2 := "ST10_RecipeDB".ParameterElement.R2GripperFixtureCode[3])
      { S7_Templates := "SrcType := String" } NE_Contact(in1 := "AutoProcessData".GripperCode_R2[3], in2 := '')
      Coil( "Robot_DB".Robot_2.GripCompareCodeOK_3 )
   END_RUNG
   RUNG wire#w1
      { S7_Templates := "SrcType := String" } EQ_Contact(in1 := "AutoProcessData".GripperCode_R2[4], in2 := "ST10_RecipeDB".ParameterElement.R2GripperFixtureCode[4])
      { S7_Templates := "SrcType := String" } NE_Contact(in1 := "AutoProcessData".GripperCode_R2[4], in2 := '')
      Coil( "Robot_DB".Robot_2.GripCompareCodeOK_4 )
   END_RUNG
   RUNG wire#w1
      Contact( "Robot_DB".Robot_2.GripCompareCodeOK_1 )
      Contact( "Robot_DB".Robot_2.GripCompareCodeOK_2 )
      Contact( "Robot_DB".Robot_2.GripCompareCodeOK_3 )
      Contact( "Robot_DB".Robot_2.GripCompareCodeOK_4 )
      Coil( "Robot_DB".Robot_2.GripCompareCodeOK )
   END_RUNG
   // the same network as SCL:
   "Robot_DB".Robot_2.GripCompareCodeOK_1 := "AlwaysTRUE" AND ("AutoProcessData".GripperCode_R2[1] = "ST10_RecipeDB".ParameterElement.R2GripperFixtureCode[1]) AND ("AutoProcessData".GripperCode_R2[1] <> '');
   "Robot_DB".Robot_2.GripCompareCodeOK_2 := "AlwaysTRUE" AND ("AutoProcessData".GripperCode_R2[2] = "ST10_RecipeDB".ParameterElement.R2GripperFixtureCode[2]) AND ("AutoProcessData".GripperCode_R2[2] <> '');
   "Robot_DB".Robot_2.GripCompareCodeOK_3 := "AlwaysTRUE" AND ("AutoProcessData".GripperCode_R2[3] = "ST10_RecipeDB".ParameterElement.R2GripperFixtureCode[3]) AND ("AutoProcessData".GripperCode_R2[3] <> '');
   "Robot_DB".Robot_2.GripCompareCodeOK_4 := "AlwaysTRUE" AND ("AutoProcessData".GripperCode_R2[4] = "ST10_RecipeDB".ParameterElement.R2GripperFixtureCode[4]) AND ("AutoProcessData".GripperCode_R2[4] <> '');
   "Robot_DB".Robot_2.GripCompareCodeOK := "AlwaysTRUE" AND "Robot_DB".Robot_2.GripCompareCodeOK_1 AND "Robot_DB".Robot_2.GripCompareCodeOK_2 AND "Robot_DB".Robot_2.GripCompareCodeOK_3 AND "Robot_DB".Robot_2.GripCompareCodeOK_4;
END_REGION

REGION Network 24: SpeedCount
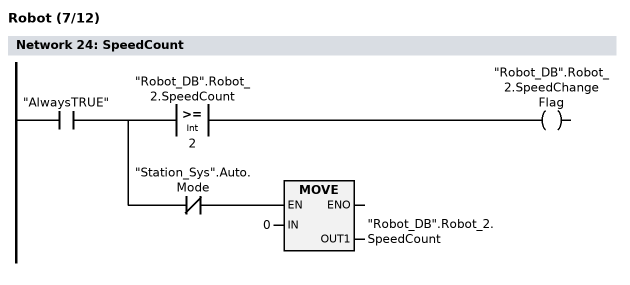
   RUNG wire#powerrail
      Contact( "AlwaysTRUE" )
      wire#w1
      { S7_Templates := "SrcType := Int" } GE_Contact(in1 := "Robot_DB".Robot_2.SpeedCount, in2 := 2)
      Coil( "Robot_DB".Robot_2.SpeedChangeFlag )
   END_RUNG
   RUNG wire#w1
      I_Contact( "Station_Sys".Auto.Mode )
      Move(in := 0, out1 => "Robot_DB".Robot_2.SpeedCount)
   END_RUNG
   // the same network as SCL:
   "Robot_DB".Robot_2.SpeedChangeFlag := "AlwaysTRUE" AND ("Robot_DB".Robot_2.SpeedCount >= 2);
   IF "AlwaysTRUE" AND NOT "Station_Sys".Auto.Mode THEN "Robot_DB".Robot_2.SpeedCount := 0; END_IF;
END_REGION

REGION Network 25: Robot2Speed Interlock
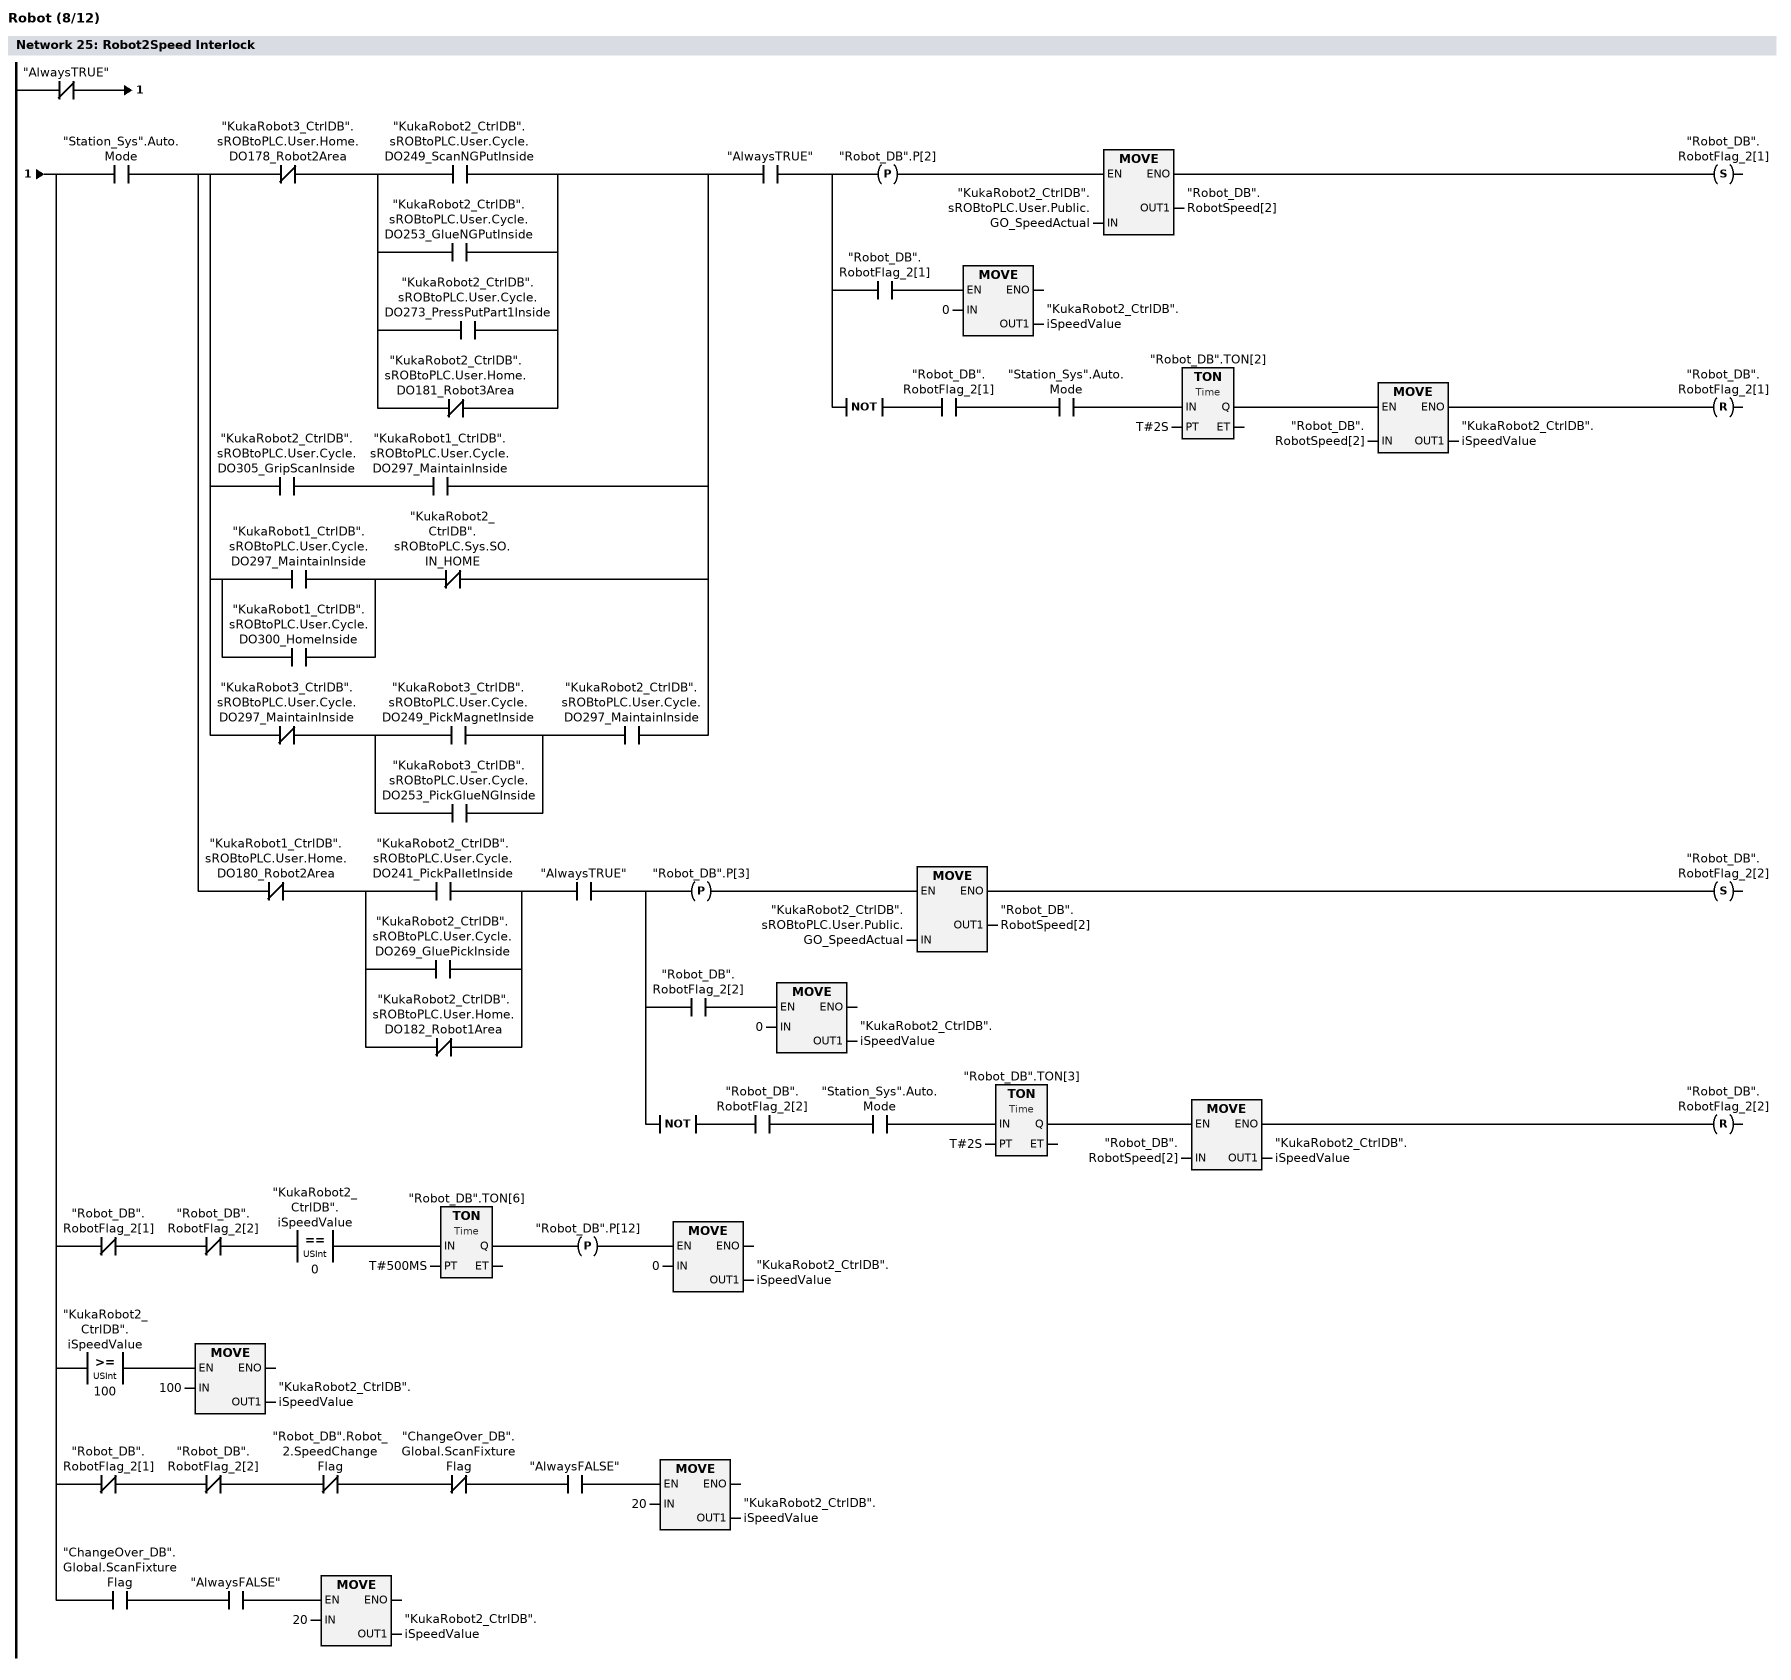
   RUNG wire#powerrail
      I_Contact( "AlwaysTRUE" )
      wire#w1
      Contact( "Station_Sys".Auto.Mode )
      wire#w2
      I_Contact( "KukaRobot3_CtrlDB".sROBtoPLC.User.Home.DO178_Robot2Area )
      wire#w3
      Contact( "KukaRobot2_CtrlDB".sROBtoPLC.User.Cycle.DO249_ScanNGPutInside )
      wire#w4
      Contact( "AlwaysTRUE" )
      wire#w8
      P_Trig( "Robot_DB".P[2] )
      Move(in := "KukaRobot2_CtrlDB".sROBtoPLC.User.Public.GO_SpeedActual, out1 => "Robot_DB".RobotSpeed[2])
      S_Coil( "Robot_DB".RobotFlag_2[1] )
   END_RUNG
   RUNG wire#w3
      Contact( "KukaRobot2_CtrlDB".sROBtoPLC.User.Cycle.DO253_GlueNGPutInside )
   END_RUNG wire#w4
   RUNG wire#w3
      Contact( "KukaRobot2_CtrlDB".sROBtoPLC.User.Cycle.DO273_PressPutPart1Inside )
   END_RUNG wire#w4
   RUNG wire#w3
      I_Contact( "KukaRobot2_CtrlDB".sROBtoPLC.User.Home.DO181_Robot3Area )
   END_RUNG wire#w4
   RUNG wire#w2
      Contact( "KukaRobot2_CtrlDB".sROBtoPLC.User.Cycle.DO305_GripScanInside )
      Contact( "KukaRobot1_CtrlDB".sROBtoPLC.User.Cycle.DO297_MaintainInside )
   END_RUNG wire#w4
   RUNG wire#w2
      Contact( "KukaRobot1_CtrlDB".sROBtoPLC.User.Cycle.DO297_MaintainInside )
      wire#w5
      I_Contact( "KukaRobot2_CtrlDB".sROBtoPLC.Sys.SO.IN_HOME )
   END_RUNG wire#w4
   RUNG wire#w2
      Contact( "KukaRobot1_CtrlDB".sROBtoPLC.User.Cycle.DO300_HomeInside )
   END_RUNG wire#w5
   RUNG wire#w2
      I_Contact( "KukaRobot3_CtrlDB".sROBtoPLC.User.Cycle.DO297_MaintainInside )
      wire#w6
      Contact( "KukaRobot3_CtrlDB".sROBtoPLC.User.Cycle.DO249_PickMagnetInside )
      wire#w7
      Contact( "KukaRobot2_CtrlDB".sROBtoPLC.User.Cycle.DO297_MaintainInside )
   END_RUNG wire#w4
   RUNG wire#w6
      Contact( "KukaRobot3_CtrlDB".sROBtoPLC.User.Cycle.DO253_PickGlueNGInside )
   END_RUNG wire#w7
   RUNG wire#w8
      Contact( "Robot_DB".RobotFlag_2[1] )
      Move(in := 0, out1 => "KukaRobot2_CtrlDB".iSpeedValue)
   END_RUNG
   RUNG wire#w8
      Not()
      Contact( "Robot_DB".RobotFlag_2[1] )
      Contact( "Station_Sys".Auto.Mode )
      { S7_Templates := "time_type := Time" } "Robot_DB".TON[2].TON(pt := T#2S, et =>)
      Move(in := "Robot_DB".RobotSpeed[2], out1 => "KukaRobot2_CtrlDB".iSpeedValue)
      R_Coil( "Robot_DB".RobotFlag_2[1] )
   END_RUNG
   RUNG wire#w2
      I_Contact( "KukaRobot1_CtrlDB".sROBtoPLC.User.Home.DO180_Robot2Area )
      wire#w9
      Contact( "KukaRobot2_CtrlDB".sROBtoPLC.User.Cycle.DO241_PickPalletInside )
      wire#w10
      Contact( "AlwaysTRUE" )
      wire#w11
      P_Trig( "Robot_DB".P[3] )
      Move(in := "KukaRobot2_CtrlDB".sROBtoPLC.User.Public.GO_SpeedActual, out1 => "Robot_DB".RobotSpeed[2])
      S_Coil( "Robot_DB".RobotFlag_2[2] )
   END_RUNG
   RUNG wire#w9
      Contact( "KukaRobot2_CtrlDB".sROBtoPLC.User.Cycle.DO269_GluePickInside )
   END_RUNG wire#w10
   RUNG wire#w9
      I_Contact( "KukaRobot2_CtrlDB".sROBtoPLC.User.Home.DO182_Robot1Area )
   END_RUNG wire#w10
   RUNG wire#w11
      Contact( "Robot_DB".RobotFlag_2[2] )
      Move(in := 0, out1 => "KukaRobot2_CtrlDB".iSpeedValue)
   END_RUNG
   RUNG wire#w11
      Not()
      Contact( "Robot_DB".RobotFlag_2[2] )
      Contact( "Station_Sys".Auto.Mode )
      { S7_Templates := "time_type := Time" } "Robot_DB".TON[3].TON(pt := T#2S, et =>)
      Move(in := "Robot_DB".RobotSpeed[2], out1 => "KukaRobot2_CtrlDB".iSpeedValue)
      R_Coil( "Robot_DB".RobotFlag_2[2] )
   END_RUNG
   RUNG wire#w1
      I_Contact( "Robot_DB".RobotFlag_2[1] )
      I_Contact( "Robot_DB".RobotFlag_2[2] )
      { S7_Templates := "SrcType := USInt" } EQ_Contact(in1 := "KukaRobot2_CtrlDB".iSpeedValue, in2 := 0)
      { S7_Templates := "time_type := Time" } "Robot_DB".TON[6].TON(pt := T#500MS, et =>)
      P_Trig( "Robot_DB".P[12] )
      Move(in := 0, out1 => "KukaRobot2_CtrlDB".iSpeedValue)
   END_RUNG
   RUNG wire#w1
      { S7_Templates := "SrcType := USInt" } GE_Contact(in1 := "KukaRobot2_CtrlDB".iSpeedValue, in2 := 100)
      Move(in := 100, out1 => "KukaRobot2_CtrlDB".iSpeedValue)
   END_RUNG
   RUNG wire#w1
      I_Contact( "Robot_DB".RobotFlag_2[1] )
      I_Contact( "Robot_DB".RobotFlag_2[2] )
      I_Contact( "Robot_DB".Robot_2.SpeedChangeFlag )
      I_Contact( "ChangeOver_DB".Global.ScanFixtureFlag )
      Contact( "AlwaysFALSE" )
      Move(in := 20, out1 => "KukaRobot2_CtrlDB".iSpeedValue)
   END_RUNG
   RUNG wire#w1
      Contact( "ChangeOver_DB".Global.ScanFixtureFlag )
      Contact( "AlwaysFALSE" )
      Move(in := 20, out1 => "KukaRobot2_CtrlDB".iSpeedValue)
   END_RUNG
   // the same network as SCL:
   #_w1 := NOT "AlwaysTRUE" AND "Station_Sys".Auto.Mode;
   #_w2 := #_w1 AND ((NOT "KukaRobot3_CtrlDB".sROBtoPLC.User.Home.DO178_Robot2Area AND ("KukaRobot2_CtrlDB".sROBtoPLC.User.Cycle.DO249_ScanNGPutInside OR "KukaRobot2_CtrlDB".sROBtoPLC.User.Cycle.DO253_GlueNGPutInside OR "KukaRobot2_CtrlDB".sROBtoPLC.User.Cycle.DO273_PressPutPart1Inside OR NOT "KukaRobot2_CtrlDB".sROBtoPLC.User.Home.DO181_Robot3Area)) OR ("KukaRobot2_CtrlDB".sROBtoPLC.User.Cycle.DO305_GripScanInside AND "KukaRobot1_CtrlDB".sROBtoPLC.User.Cycle.DO297_MaintainInside) OR (("KukaRobot1_CtrlDB".sROBtoPLC.User.Cycle.DO297_MaintainInside OR "KukaRobot1_CtrlDB".sROBtoPLC.User.Cycle.DO300_HomeInside) AND NOT "KukaRobot2_CtrlDB".sROBtoPLC.Sys.SO.IN_HOME) OR (NOT "KukaRobot3_CtrlDB".sROBtoPLC.User.Cycle.DO297_MaintainInside AND ("KukaRobot3_CtrlDB".sROBtoPLC.User.Cycle.DO249_PickMagnetInside OR "KukaRobot3_CtrlDB".sROBtoPLC.User.Cycle.DO253_PickGlueNGInside) AND "KukaRobot2_CtrlDB".sROBtoPLC.User.Cycle.DO297_MaintainInside)) AND "AlwaysTRUE";
   #_w3 := #_w2 AND NOT "Robot_DB".P[2];   // rising edge
   "Robot_DB".P[2] := #_w2;
   IF #_w3 THEN
       "Robot_DB".RobotSpeed[2] := "KukaRobot2_CtrlDB".sROBtoPLC.User.Public.GO_SpeedActual;
       "Robot_DB".RobotFlag_2[1] := TRUE;
   END_IF;
   IF #_w2 AND "Robot_DB".RobotFlag_2[1] THEN "KukaRobot2_CtrlDB".iSpeedValue := 0; END_IF;
   "Robot_DB".TON[2].TON(IN := NOT #_w2 AND "Robot_DB".RobotFlag_2[1] AND "Station_Sys".Auto.Mode, PT := T#2S);
   IF "Robot_DB".TON[2].Q THEN
       "KukaRobot2_CtrlDB".iSpeedValue := "Robot_DB".RobotSpeed[2];
       "Robot_DB".RobotFlag_2[1] := FALSE;
   END_IF;
   #_w4 := #_w1 AND NOT "KukaRobot1_CtrlDB".sROBtoPLC.User.Home.DO180_Robot2Area AND ("KukaRobot2_CtrlDB".sROBtoPLC.User.Cycle.DO241_PickPalletInside OR "KukaRobot2_CtrlDB".sROBtoPLC.User.Cycle.DO269_GluePickInside OR NOT "KukaRobot2_CtrlDB".sROBtoPLC.User.Home.DO182_Robot1Area) AND "AlwaysTRUE";
   #_w5 := #_w4 AND NOT "Robot_DB".P[3];   // rising edge
   "Robot_DB".P[3] := #_w4;
   IF #_w5 THEN
       "Robot_DB".RobotSpeed[2] := "KukaRobot2_CtrlDB".sROBtoPLC.User.Public.GO_SpeedActual;
       "Robot_DB".RobotFlag_2[2] := TRUE;
   END_IF;
   IF #_w4 AND "Robot_DB".RobotFlag_2[2] THEN "KukaRobot2_CtrlDB".iSpeedValue := 0; END_IF;
   "Robot_DB".TON[3].TON(IN := NOT #_w4 AND "Robot_DB".RobotFlag_2[2] AND "Station_Sys".Auto.Mode, PT := T#2S);
   IF "Robot_DB".TON[3].Q THEN
       "KukaRobot2_CtrlDB".iSpeedValue := "Robot_DB".RobotSpeed[2];
       "Robot_DB".RobotFlag_2[2] := FALSE;
   END_IF;
   "Robot_DB".TON[6].TON(IN := NOT "AlwaysTRUE" AND NOT "Robot_DB".RobotFlag_2[1] AND NOT "Robot_DB".RobotFlag_2[2] AND ("KukaRobot2_CtrlDB".iSpeedValue = 0),
                         PT := T#500MS);
   #_w6 := "Robot_DB".TON[6].Q AND NOT "Robot_DB".P[12];   // rising edge
   "Robot_DB".P[12] := "Robot_DB".TON[6].Q;
   IF #_w6 THEN "KukaRobot2_CtrlDB".iSpeedValue := 0; END_IF;
   IF NOT "AlwaysTRUE" AND ("KukaRobot2_CtrlDB".iSpeedValue >= 100) THEN
       "KukaRobot2_CtrlDB".iSpeedValue := 100;
   END_IF;
   IF NOT "AlwaysTRUE" AND NOT "Robot_DB".RobotFlag_2[1] AND NOT "Robot_DB".RobotFlag_2[2] AND NOT "Robot_DB".Robot_2.SpeedChangeFlag AND NOT "ChangeOver_DB".Global.ScanFixtureFlag AND "AlwaysFALSE" THEN
       "KukaRobot2_CtrlDB".iSpeedValue := 20;
   END_IF;
   IF NOT "AlwaysTRUE" AND "ChangeOver_DB".Global.ScanFixtureFlag AND "AlwaysFALSE" THEN
       "KukaRobot2_CtrlDB".iSpeedValue := 20;
   END_IF;
END_REGION

REGION Network 26: Robot2 No Task Running
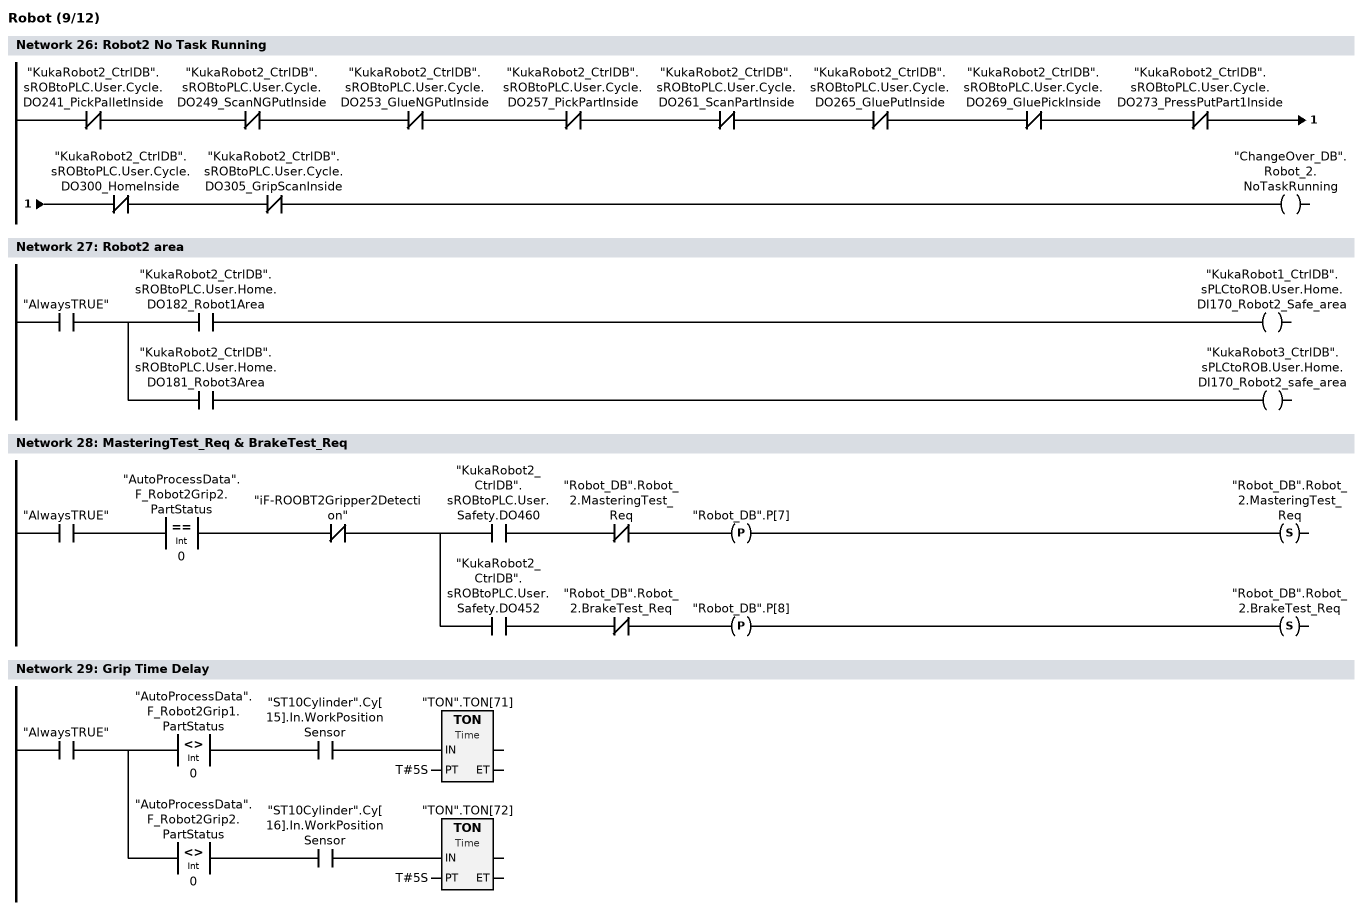
   RUNG wire#powerrail
      I_Contact( "KukaRobot2_CtrlDB".sROBtoPLC.User.Cycle.DO241_PickPalletInside )
      I_Contact( "KukaRobot2_CtrlDB".sROBtoPLC.User.Cycle.DO249_ScanNGPutInside )
      I_Contact( "KukaRobot2_CtrlDB".sROBtoPLC.User.Cycle.DO253_GlueNGPutInside )
      I_Contact( "KukaRobot2_CtrlDB".sROBtoPLC.User.Cycle.DO257_PickPartInside )
      I_Contact( "KukaRobot2_CtrlDB".sROBtoPLC.User.Cycle.DO261_ScanPartInside )
      I_Contact( "KukaRobot2_CtrlDB".sROBtoPLC.User.Cycle.DO265_GluePutInside )
      I_Contact( "KukaRobot2_CtrlDB".sROBtoPLC.User.Cycle.DO269_GluePickInside )
      I_Contact( "KukaRobot2_CtrlDB".sROBtoPLC.User.Cycle.DO273_PressPutPart1Inside )
      I_Contact( "KukaRobot2_CtrlDB".sROBtoPLC.User.Cycle.DO300_HomeInside )
      I_Contact( "KukaRobot2_CtrlDB".sROBtoPLC.User.Cycle.DO305_GripScanInside )
      Coil( "ChangeOver_DB".Robot_2.NoTaskRunning )
   END_RUNG
   // the same network as SCL:
   "ChangeOver_DB".Robot_2.NoTaskRunning := NOT "KukaRobot2_CtrlDB".sROBtoPLC.User.Cycle.DO241_PickPalletInside AND NOT "KukaRobot2_CtrlDB".sROBtoPLC.User.Cycle.DO249_ScanNGPutInside AND NOT "KukaRobot2_CtrlDB".sROBtoPLC.User.Cycle.DO253_GlueNGPutInside AND NOT "KukaRobot2_CtrlDB".sROBtoPLC.User.Cycle.DO257_PickPartInside AND NOT "KukaRobot2_CtrlDB".sROBtoPLC.User.Cycle.DO261_ScanPartInside AND NOT "KukaRobot2_CtrlDB".sROBtoPLC.User.Cycle.DO265_GluePutInside AND NOT "KukaRobot2_CtrlDB".sROBtoPLC.User.Cycle.DO269_GluePickInside AND NOT "KukaRobot2_CtrlDB".sROBtoPLC.User.Cycle.DO273_PressPutPart1Inside AND NOT "KukaRobot2_CtrlDB".sROBtoPLC.User.Cycle.DO300_HomeInside AND NOT "KukaRobot2_CtrlDB".sROBtoPLC.User.Cycle.DO305_GripScanInside;
END_REGION

REGION Network 27: Robot2 area
   RUNG wire#powerrail
      Contact( "AlwaysTRUE" )
      wire#w1
      Contact( "KukaRobot2_CtrlDB".sROBtoPLC.User.Home.DO182_Robot1Area )
      Coil( "KukaRobot1_CtrlDB".sPLCtoROB.User.Home.DI170_Robot2_Safe_area )
   END_RUNG
   RUNG wire#w1
      Contact( "KukaRobot2_CtrlDB".sROBtoPLC.User.Home.DO181_Robot3Area )
      Coil( "KukaRobot3_CtrlDB".sPLCtoROB.User.Home.DI170_Robot2_safe_area )
   END_RUNG
   // the same network as SCL:
   "KukaRobot1_CtrlDB".sPLCtoROB.User.Home.DI170_Robot2_Safe_area := "AlwaysTRUE" AND "KukaRobot2_CtrlDB".sROBtoPLC.User.Home.DO182_Robot1Area;
   "KukaRobot3_CtrlDB".sPLCtoROB.User.Home.DI170_Robot2_safe_area := "AlwaysTRUE" AND "KukaRobot2_CtrlDB".sROBtoPLC.User.Home.DO181_Robot3Area;
END_REGION

REGION Network 28: MasteringTest_Req & BrakeTest_Req
   RUNG wire#powerrail
      Contact( "AlwaysTRUE" )
      { S7_Templates := "SrcType := Int" } EQ_Contact(in1 := "AutoProcessData".F_Robot2Grip2.PartStatus, in2 := 0)
      I_Contact( "iF-ROOBT2Gripper2Detection" )
      wire#w1
      Contact( "KukaRobot2_CtrlDB".sROBtoPLC.User.Safety.DO460 )
      I_Contact( "Robot_DB".Robot_2.MasteringTest_Req )
      P_Trig( "Robot_DB".P[7] )
      S_Coil( "Robot_DB".Robot_2.MasteringTest_Req )
   END_RUNG
   RUNG wire#w1
      Contact( "KukaRobot2_CtrlDB".sROBtoPLC.User.Safety.DO452 )
      I_Contact( "Robot_DB".Robot_2.BrakeTest_Req )
      P_Trig( "Robot_DB".P[8] )
      S_Coil( "Robot_DB".Robot_2.BrakeTest_Req )
   END_RUNG
   // the same network as SCL:
   #_w1 := "AlwaysTRUE" AND ("AutoProcessData".F_Robot2Grip2.PartStatus = 0) AND NOT "iF-ROOBT2Gripper2Detection";
   #_w2 := #_w1 AND "KukaRobot2_CtrlDB".sROBtoPLC.User.Safety.DO460 AND NOT "Robot_DB".Robot_2.MasteringTest_Req;
   #_w3 := #_w2 AND NOT "Robot_DB".P[7];   // rising edge
   "Robot_DB".P[7] := #_w2;
   IF #_w3 THEN "Robot_DB".Robot_2.MasteringTest_Req := TRUE; END_IF;
   #_w4 := #_w1 AND "KukaRobot2_CtrlDB".sROBtoPLC.User.Safety.DO452 AND NOT "Robot_DB".Robot_2.BrakeTest_Req;
   #_w5 := #_w4 AND NOT "Robot_DB".P[8];   // rising edge
   "Robot_DB".P[8] := #_w4;
   IF #_w5 THEN "Robot_DB".Robot_2.BrakeTest_Req := TRUE; END_IF;
END_REGION

REGION Network 29: Grip Time Delay
   RUNG wire#powerrail
      Contact( "AlwaysTRUE" )
      wire#w1
      { S7_Templates := "SrcType := Int" } NE_Contact(in1 := "AutoProcessData".F_Robot2Grip1.PartStatus, in2 := 0)
      Contact( "ST10Cylinder".Cy[15].In.WorkPositionSensor )
      { S7_Templates := "time_type := Time" } "TON".TON[71].TON(pt := T#5S, et =>)
   END_RUNG
   RUNG wire#w1
      { S7_Templates := "SrcType := Int" } NE_Contact(in1 := "AutoProcessData".F_Robot2Grip2.PartStatus, in2 := 0)
      Contact( "ST10Cylinder".Cy[16].In.WorkPositionSensor )
      { S7_Templates := "time_type := Time" } "TON".TON[72].TON(pt := T#5S, et =>)
   END_RUNG
   // the same network as SCL:
   "TON".TON[71].TON(IN := "AlwaysTRUE" AND ("AutoProcessData".F_Robot2Grip1.PartStatus <> 0) AND "ST10Cylinder".Cy[15].In.WorkPositionSensor,
                     PT := T#5S);
   "TON".TON[72].TON(IN := "AlwaysTRUE" AND ("AutoProcessData".F_Robot2Grip2.PartStatus <> 0) AND "ST10Cylinder".Cy[16].In.WorkPositionSensor,
                     PT := T#5S);
END_REGION

REGION Network 31: ----------------------------------------- Robot_3 -------------------------------------
END_REGION

REGION Network 32: CodeCompare
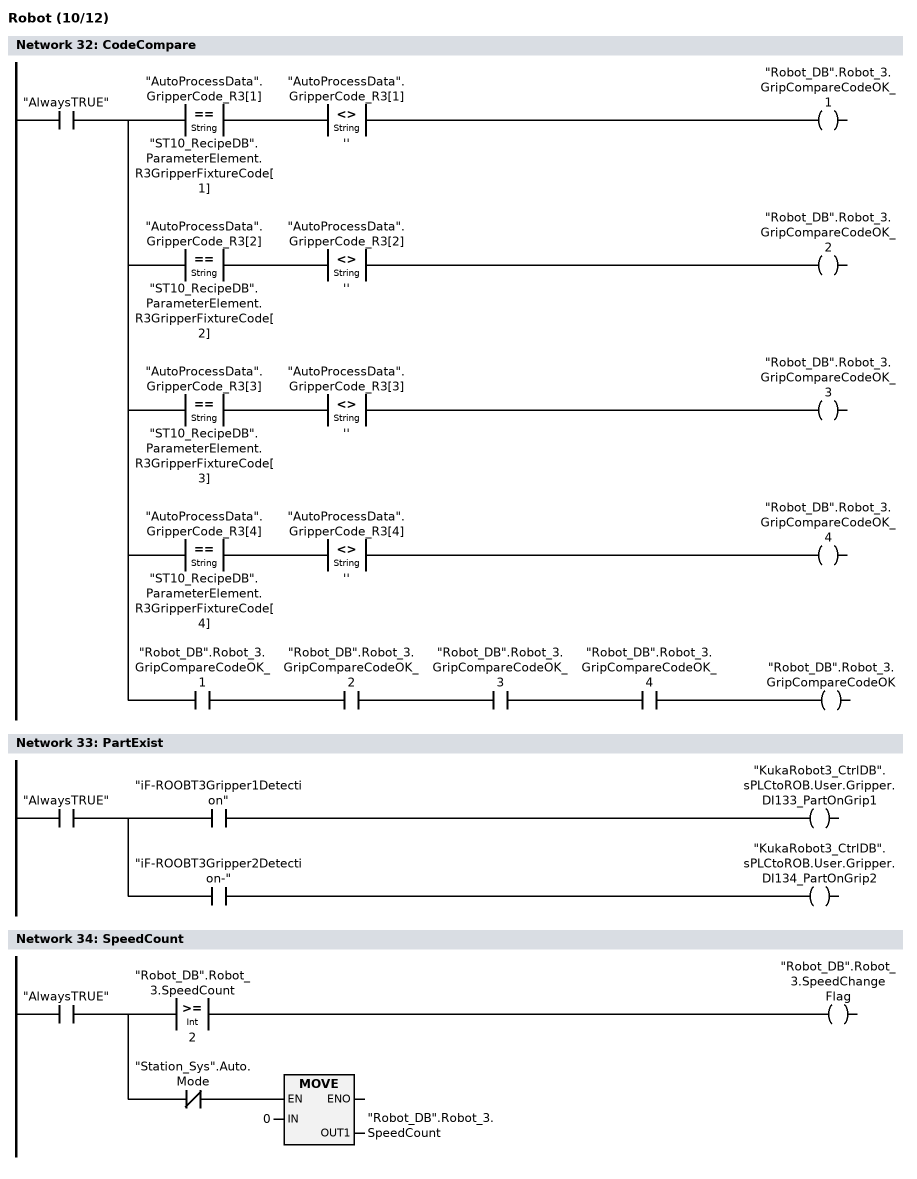
   RUNG wire#powerrail
      Contact( "AlwaysTRUE" )
      wire#w1
      { S7_Templates := "SrcType := String" } EQ_Contact(in1 := "AutoProcessData".GripperCode_R3[1], in2 := "ST10_RecipeDB".ParameterElement.R3GripperFixtureCode[1])
      { S7_Templates := "SrcType := String" } NE_Contact(in1 := "AutoProcessData".GripperCode_R3[1], in2 := '')
      Coil( "Robot_DB".Robot_3.GripCompareCodeOK_1 )
   END_RUNG
   RUNG wire#w1
      { S7_Templates := "SrcType := String" } EQ_Contact(in1 := "AutoProcessData".GripperCode_R3[2], in2 := "ST10_RecipeDB".ParameterElement.R3GripperFixtureCode[2])
      { S7_Templates := "SrcType := String" } NE_Contact(in1 := "AutoProcessData".GripperCode_R3[2], in2 := '')
      Coil( "Robot_DB".Robot_3.GripCompareCodeOK_2 )
   END_RUNG
   RUNG wire#w1
      { S7_Templates := "SrcType := String" } EQ_Contact(in1 := "AutoProcessData".GripperCode_R3[3], in2 := "ST10_RecipeDB".ParameterElement.R3GripperFixtureCode[3])
      { S7_Templates := "SrcType := String" } NE_Contact(in1 := "AutoProcessData".GripperCode_R3[3], in2 := '')
      Coil( "Robot_DB".Robot_3.GripCompareCodeOK_3 )
   END_RUNG
   RUNG wire#w1
      { S7_Templates := "SrcType := String" } EQ_Contact(in1 := "AutoProcessData".GripperCode_R3[4], in2 := "ST10_RecipeDB".ParameterElement.R3GripperFixtureCode[4])
      { S7_Templates := "SrcType := String" } NE_Contact(in1 := "AutoProcessData".GripperCode_R3[4], in2 := '')
      Coil( "Robot_DB".Robot_3.GripCompareCodeOK_4 )
   END_RUNG
   RUNG wire#w1
      Contact( "Robot_DB".Robot_3.GripCompareCodeOK_1 )
      Contact( "Robot_DB".Robot_3.GripCompareCodeOK_2 )
      Contact( "Robot_DB".Robot_3.GripCompareCodeOK_3 )
      Contact( "Robot_DB".Robot_3.GripCompareCodeOK_4 )
      Coil( "Robot_DB".Robot_3.GripCompareCodeOK )
   END_RUNG
   // the same network as SCL:
   "Robot_DB".Robot_3.GripCompareCodeOK_1 := "AlwaysTRUE" AND ("AutoProcessData".GripperCode_R3[1] = "ST10_RecipeDB".ParameterElement.R3GripperFixtureCode[1]) AND ("AutoProcessData".GripperCode_R3[1] <> '');
   "Robot_DB".Robot_3.GripCompareCodeOK_2 := "AlwaysTRUE" AND ("AutoProcessData".GripperCode_R3[2] = "ST10_RecipeDB".ParameterElement.R3GripperFixtureCode[2]) AND ("AutoProcessData".GripperCode_R3[2] <> '');
   "Robot_DB".Robot_3.GripCompareCodeOK_3 := "AlwaysTRUE" AND ("AutoProcessData".GripperCode_R3[3] = "ST10_RecipeDB".ParameterElement.R3GripperFixtureCode[3]) AND ("AutoProcessData".GripperCode_R3[3] <> '');
   "Robot_DB".Robot_3.GripCompareCodeOK_4 := "AlwaysTRUE" AND ("AutoProcessData".GripperCode_R3[4] = "ST10_RecipeDB".ParameterElement.R3GripperFixtureCode[4]) AND ("AutoProcessData".GripperCode_R3[4] <> '');
   "Robot_DB".Robot_3.GripCompareCodeOK := "AlwaysTRUE" AND "Robot_DB".Robot_3.GripCompareCodeOK_1 AND "Robot_DB".Robot_3.GripCompareCodeOK_2 AND "Robot_DB".Robot_3.GripCompareCodeOK_3 AND "Robot_DB".Robot_3.GripCompareCodeOK_4;
END_REGION

